(* CODESYS project Full_Project.export

Project tree, tasks and I/O mapping:
  CODESYS_Control_x86_Arca_Control_SM : CODESYS Control x86 Arca Control SM, 3S - Smart Software Solutions GmbH, version 3.5.8.0
    application Application
      libraries: Standard, * (System); Arca Motion Library, 1.0.4.14 (BonMET); Network, 3.5.7.0 (3S - Smart Software Solutions GmbH)
      task Task (cyclic, interval t#5ms, priority 1) calls Main
      AxisControl/
        data type MutiAxisMoveMethod
        function block AuxAxis_PowerOn [ST]
        function block MultiAxisABSMove [ST]
        function block MultiAxisTorqueLimit [ST]
      Hand_Control_blocks/
        data type Error_Message
        data type Gesture_Type
        data type Grab_Command
        data type Grab_State
        data type PhysicalHandType
        function block Grab_Control [ST]
        function block Grab_Demo [ST]
        function block Hand_Gesture [ST]
        function block Hand_Gesture_Demo [ST]
      IO_Management/
        function block Digital_Input [ST]
        function block Digital_Input_Analog [ST]
        function block Digital_Output [ST]
      TCPIP Control/
        data type Robot_Command_via_tcp
        data type Robot_State
        function block TCPServerConnection [ST]
        function block TCP_Command_Extract_And_Analysis [ST]
      Testment_Cartesian_Laser_Platform_Test/
        program Cartesian_Laser_Circle_Testment [ST]
      Testment_Servo_Function_Test/
        program Servo_Testment_Main [ST]
        function block Testment_Message_Manager [ST]
      Utility_functions/
        function block Value_Clamp [ST]
      global variables GLobal_Value
      program Cartesin [ST]
      program Main [ST]
      program Read_Basic_Info [ST]
      program SingleAxis [ST]
    SoftMotion General Axis Pool
*)

// CODESYS_Control_x86_Arca_Control_SM/Application/AxisControl/MutiAxisMoveMethod
TYPE MutiAxisMoveMethod :
(
	None := 0				// all axis move at same vel as given
	, SpeedControl := 10		// all axis arrive destination at same time
);
END_TYPE

// CODESYS_Control_x86_Arca_Control_SM/Application/Hand_Control_blocks/Error_Message
{attribute 'qualified_only'}
{attribute 'strict'}
TYPE Error_Message :
(
	Err_None := 0,
	
	Err_AuxAxis_Movement_Cannot_read_virture_robot_position := 10,	// gesture block not reading robot position
	Err_Gesture_Type_Hand_Pos_Not_Given := 20,	// gesture block not given position
	Err_AuxAxis_Movement_Block_err := 30,	// gesture block first reset movement block err
	Err_Gesture_Type_Cycle_mov_block_err := 40,	// gesture block cycle movement block err
	
	Err_PowerOn_Block_Err := 50,
	Err_PowerOn_TimeOut := 51,
	
	Err_Power_Reset_Block_Err := 60,
	Err_Power_Reset_TimeOut := 61,
	
	Err_Group_Enable_Block_Err := 70,
	Err_Group_Enable_TimeOut := 71
);
END_TYPE

// CODESYS_Control_x86_Arca_Control_SM/Application/Hand_Control_blocks/Gesture_Type
{attribute 'qualified_only'}
{attribute 'strict'}
TYPE Gesture_Type :
(
	Gesture_Type_None			:= 0,
	Gesture_Type_Num_1		:= 1,
	Gesture_Type_Num_2		:= 2,
	Gesture_Type_Num_3		:= 3,
	Gesture_Type_Num_4		:= 4,
	Gesture_Type_Num_5		:= 5,
	Gesture_Type_Num_6		:= 6,
	Gesture_Type_Fist			:= 10,
	Gesture_Type_Palm			:= 11,
	Gesture_Type_ThumbUp		:= 12,
	Gesture_Type_NoNoNo			:= 13,
	Gesture_Type_ComeOnBaby	:= 14,
	Gesture_Type_FingerWave		:= 15,
	Gesture_Type_Wave			:= 16,
	Gesture_Type_Nya			:= 17,
	Gesture_Type_MovObj			:= 18
);
END_TYPE

// CODESYS_Control_x86_Arca_Control_SM/Application/Hand_Control_blocks/Grab_Command
TYPE Grab_Command :
STRUCT
	Tip_Angle : REAL;
	Root_Angle : REAL;
	Clamp_Angle : REAL;
END_STRUCT
END_TYPE

// CODESYS_Control_x86_Arca_Control_SM/Application/Hand_Control_blocks/Grab_State
TYPE Grab_State :
STRUCT
	Tip_State : BOOL;
	Root_State : BOOL;
	Clamp_Angle : REAL;
END_STRUCT
END_TYPE

// CODESYS_Control_x86_Arca_Control_SM/Application/Hand_Control_blocks/PhysicalHandType
TYPE PhysicalHandType :
(
	motor18		:= 0	// total 18 motors. 4 axis for thumb, 3 axis control 2 joints, anohter one control thumb tip joint. Other fingers has 3 axis each, each axis control 1 jonit. 2 axis for each wrist joint.
	, motor17	:= 10	// total 17 motors, each axis control 1 joint.
);
END_TYPE

// CODESYS_Control_x86_Arca_Control_SM/Application/TCPIP Control/Robot_Command_via_tcp
TYPE Robot_Command_via_tcp :
STRUCT
	X_Axis_Valid : BOOL;
	X_value : REAL;
	Y_Axis_Valid : BOOL;
	Y_value : REAL;
	Z_Axis_Valid : BOOL;
	Z_value : REAL;
	Spin : BOOL;
	Grab_Valid : BOOL;
	Grab_state : BOOL := FALSE;
	Gesture_Valid : BOOL;
	Gesture_Num : Gesture_Type;
	Enabl_Hand_Valid : BOOL;
	Enabl_Hand_state : BOOL;
	Gesture_Demo_Valid : BOOL;
	Gesture_Demo_state : BOOL;
	CNC_Mov_Valid : BOOL;
	CNC_Mov_Program_Num : INT;
END_STRUCT
END_TYPE

// CODESYS_Control_x86_Arca_Control_SM/Application/TCPIP Control/Robot_State
TYPE Robot_State :
STRUCT
	Hand_Enabled : BOOL;
	Hand_Enb_Err : BOOL;
	Grab_State : BOOL;
	Gesture_State : Gesture_Type := gesture_type.Gesture_Type_None;
	Hand_Mov_Err : BOOL;
	Robot_Mov_Err : BOOL;
	CNC_Executing : BOOL;
	CNC_Execute_Done : BOOL;
	CNC_Execute_Err : BOOL;
END_STRUCT
END_TYPE

// CODESYS_Control_x86_Arca_Control_SM/Application/GLobal_Value
VAR_GLOBAL
	AllAxisGroupEnb : BOOL;
	Num_of_Axis_GV:WORD;
	Num_of_Groups_GV:WORD;
	Num_of_Cams_GV:WORD;
	MotionCfgOK_GV: BOOL;
	ECatCfgOk_GV: BOOL;
	VisionCfgOk_GV: BOOL;
END_VAR

// CODESYS_Control_x86_Arca_Control_SM/Application/Main
PROGRAM Main
VAR
END_VAR

Read_Basic_Info();

SingleAxis();

Cartesin();

Servo_Testment_Main();

END_PROGRAM

// CODESYS_Control_x86_Arca_Control_SM/Application/Read_Basic_Info
PROGRAM Read_Basic_Info
VAR	
	// read cfg message
	ReadCfg : ArcaLibrary.SYS_GetConfigInfo;
END_VAR

// read how many axis has been config, all *_GV value is golbal value
ReadCfg(axisnumber => Num_of_Axis_GV, groupnumber => Num_of_Groups_GV, cameranumber => Num_of_Cams_GV
	, MotionCfgOk => MotionCfgOK_GV, ecatcfgok => ECatCfgOk_GV, visioncfgok => VisionCfgOk_GV);

END_PROGRAM

// CODESYS_Control_x86_Arca_Control_SM/Application/SingleAxis
PROGRAM SingleAxis
VAR
	Enable : BOOL;
	StartMov : BOOL;
	MovAxis : INT := 0;
	FirstPos : REAL := -180;
	SecondPos : REAL := 180;
	CurrentPos : REAL;
	Vel : REAL := 180;
	Acc : REAL := 180;
	Jerk : REAL := 180;
	stopTime : TIME := T#1S;
	MovErr : BOOL;
	
	PowBlk : ArcaLibrary.MC_Power;
	PowDone, PowErr : BOOL;
	
	MovState : INT;
	FirMov : ArcaLibrary.MC_MoveAbsolute;
	SecMov : ArcaLibrary.MC_MoveAbsolute;
	StopMov : ArcaLibrary.MC_Stop;
	dis_trig : r_trig;
	
	ReadPos : ArcaLibrary.MCAT_ReadAxisMeasures;
	StopTimer : ton;
END_VAR


PowBlk(Axis := MovAxis, Enable:=Enable, EnablePositive:=TRUE, EnableNegative:=TRUE, Status=>PowDone, Error=>PowErr);
ReadPos(axis := MovAxis, enable := PowBlk.Status, pos=> currentPos);

dis_trig(clk := NOT startMov);
StopMov(axis := MovAxis, execute := dis_trig.Q, Deceleration := acc*10, jerk := jerk*10);

IF MovState > 20 AND NOT startMov THEN
	MovState := 20;
END_IF
CASE MovState OF
	0:
		IF PowDone THEN
			MovState := 10;
		END_IF
	10:
		IF startMov THEN
			MovState := 20;
		END_IF
	20:
		FirMov(axis := MovAxis, Execute := FALSE);
		SecMov(axis := MovAxis, Execute := FALSE);
		IF startMov THEN
			StopTimer(in:= FALSE);
			MovState := 30;
		ELSE
			MovState := 0;
		END_IF
	30:
		FirMov(axis := MovAxis, Execute := TRUE, Position := FirstPos
			, Velocity := vel, Acceleration := acc, Deceleration := Acc, jerk := jerk
			, Direction := mcShortestWay, BufferMode := mcAborting 
			, Error => MovErr);
		IF FirMov.Done THEN
			IF stopTime > T#0S THEN
			StopTimer (in := TRUE, PT := stopTime);
				MovState := 35;
			ELSE
				MovState := 40;
			END_IF
		END_IF
	35:
		StopTimer (in := TRUE, PT := stopTime);
		IF StopTimer.Q THEN
			StopTimer(in:= FALSE);
			MovState := 40;
		END_IF
	40:
		SecMov(axis := MovAxis, Execute := TRUE, Position := SecondPos
			, Velocity := vel, Acceleration := acc, Deceleration := Acc, jerk := jerk
			, Direction := mcShortestWay, BufferMode := mcAborting 
			, Error => MovErr);
		IF SecMov.Done THEN
			StopTimer (in := TRUE, PT := stopTime);
			IF stopTime > T#0S THEN
				MovState := 45;
			ELSE
			MovState := 20;
			END_IF
		END_IF
	45:
		StopTimer (in := TRUE, PT := stopTime);
		IF StopTimer.Q THEN
			StopTimer(in:= FALSE);
			MovState := 20;
		END_IF
END_CASE

END_PROGRAM

// CODESYS_Control_x86_Arca_Control_SM/Application/Cartesin
PROGRAM Cartesin
VAR
	Enable : BOOL;
	StartMov : BOOL;
	safe_pos :  ARRAY [1..6] OF REAL := [0.0, 0.0, 0.0, 0.0, -90.0, 0.0];
	FirstReachPos :  ARRAY [1..6] OF REAL := [0.562, 0.333, 0.606, 118.70, 167.069, -70.06];
	SecondReachPos :  ARRAY [1..6] OF REAL := [0.562, 0.3, 0.606, 118.70, 167.069, -70.06];
	FirstPerPos :  ARRAY [1..6] OF REAL := [0.562, 0.333, 0.636, 118.70, 167.069, -70.06];
	SecondPerPos :  ARRAY [1..6] OF REAL := [0.562, 0.3, 0.636, 118.70, 167.069, -70.06];
	
	CurrentPos : REAL;
	Vel : REAL := 10;
	Acc : REAL := 10;
	Jerk : REAL := 10;
	safepoint_overfeed : INT := 5; 
	GrRelCorner :REAL := 0.5;
	MovGroup : INT := 0;
	
	MovErr : BOOL;
	
	PowBlk : AuxAxis_PowerOn;
	PowDone, PowErr : BOOL;
	
	MovState : INT;
	InitialMov : ArcaLibrary.MCAT_MoveDirect;;
	Movs : ARRAY [0..6] OF ArcaLibrary.MC_MoveLinearAbsolute;
	StopMov : ArcaLibrary.MC_GroupStop;
	dis_trig : r_trig;
	
	
END_VAR

PowBlk(Enable := enable, done => PowDone);

dis_trig(clk := NOT startMov);
StopMov(AxesGroup := MovGroup, execute := dis_trig.Q, Deceleration := acc, jerk := jerk, BufferMode := mcAborting);

IF MovState > 20 AND NOT startMov THEN
	MovState := 20;
END_IF
CASE MovState OF
	0:
		IF PowDone THEN
			MovState := 10;
		END_IF
	10:
		IF startMov THEN
			MovState := 20;
		END_IF
	20:
		InitialMov(axesgroup := MovGroup, execute := FALSE);
		Movs[0](axesgroup := MovGroup, Execute := FALSE);
		Movs[1](axesgroup := MovGroup, Execute := FALSE);
		Movs[2](axesgroup := MovGroup, Execute := FALSE);
		Movs[3](axesgroup := MovGroup, Execute := FALSE);
		Movs[4](axesgroup := MovGroup, Execute := FALSE);
		Movs[5](axesgroup := MovGroup, Execute := FALSE);
		IF startMov THEN
			MovState := 30;
		ELSE
			MovState := 0;
		END_IF
	30:
		InitialMov(axesgroup := MovGroup, execute := TRUE, position := ADR(safe_pos), coordsystem := mcacs
			, BufferMode:=mcAborting, TransitionMode:= tmNone, TransitionParameter:= ADR(GrRelCorner) 
			, OverFeedPerc:= safepoint_overfeed);
		IF initialmov.Done THEN
			MovState := 40;
		END_IF
	40:
		IF Movs[4].Done THEN
			Movs[5](axesgroup := MovGroup, Execute := TRUE, Position := ADR(SecondPerPos)
				, Velocity := vel, Acceleration := acc, Deceleration := Acc, jerk := jerk
				, coordsystem := mcMcs, BufferMode := mcBlendingNext
				, TransitionMode := TMcornerdistance, TransitionParameter:=ADR(GrRelCorner)
				, Error => MovErr);
		END_IF
		Movs[0](axesgroup := MovGroup, Execute := TRUE, Position := ADR(FirstPerPos)
			, Velocity := vel, Acceleration := acc, Deceleration := Acc, jerk := jerk
			, coordsystem := mcMcs, BufferMode := mcBlendingNext
			, TransitionMode := TMcornerdistance, TransitionParameter:=ADR(GrRelCorner)
			, Error => MovErr);
		Movs[1](axesgroup := MovGroup, Execute := TRUE, Position := ADR(FirstReachPos)
			, Velocity := vel, Acceleration := acc, Deceleration := Acc, jerk := jerk
			, coordsystem := mcMcs, BufferMode := mcBlendingPrev
			, TransitionMode := TMcornerdistance, TransitionParameter:=ADR(GrRelCorner)
			, Error => MovErr);
		IF Movs[1].Done THEN
			Movs[2](axesgroup := MovGroup, Execute := FALSE);
			Movs[3](axesgroup := MovGroup, Execute := FALSE);
			Movs[4](axesgroup := MovGroup, Execute := FALSE);
			MovState := 50;
		END_IF
	50:
		Movs[2](axesgroup := MovGroup, Execute := TRUE, Position := ADR(FirstPerPos)
			, Velocity := vel, Acceleration := acc, Deceleration := Acc, jerk := jerk
			, coordsystem := mcMcs, BufferMode := mcBlendingNext
			, TransitionMode := TMcornerdistance, TransitionParameter:=ADR(GrRelCorner)
			, Error => MovErr);
		Movs[3](axesgroup := MovGroup, Execute := TRUE, Position := ADR(SecondPerPos)
			, Velocity := vel, Acceleration := acc, Deceleration := Acc, jerk := jerk
			, coordsystem := mcMcs, BufferMode := mcBlendingNext
			, TransitionMode := TMcornerdistance, TransitionParameter:=ADR(GrRelCorner)
			, Error => MovErr);
		Movs[4](axesgroup := MovGroup, Execute := TRUE, Position := ADR(SecondReachPos)
			, Velocity := vel, Acceleration := acc, Deceleration := Acc, jerk := jerk
			, coordsystem := mcMcs, BufferMode := mcBlendingPrev
			, TransitionMode := TMcornerdistance, TransitionParameter:=ADR(GrRelCorner)
			, Error => MovErr);
		IF Movs[4].Done THEN
			Movs[0](axesgroup := MovGroup, Execute := FALSE);
			Movs[1](axesgroup := MovGroup, Execute := FALSE);
			Movs[5](axesgroup := MovGroup, Execute := FALSE);
			MovState := 40;
		END_IF
END_CASE

END_PROGRAM

// CODESYS_Control_x86_Arca_Control_SM/Application/AxisControl/AuxAxis_PowerOn
FUNCTION_BLOCK AuxAxis_PowerOn
VAR_INPUT
	Enable : BOOL;
END_VAR
VAR_OUTPUT
	Done : BOOL;
	Error : BOOL;
	Err_Message : Error_Message;
END_VAR
VAR
	_state : INT := 0;
	_end : BOOL := TRUE;
	_Timer: ton;
	_err_time : TIME := T#5S;
	
	// read cfg message
	ReadCfg : ArcaLibrary.SYS_GetConfigInfo;
	Num_of_Axis:WORD;
	Num_of_Groups:WORD;
	Num_of_Cams:WORD;
	MotionCfgOK: BOOL;
	ECatCfgOk: BOOL;
	VisionCfgOk: BOOL;
	
	// power settings
	PowBlk:ARRAY[1..48] OF ArcaLibrary.MC_Power;
	PowDone, PowErr: ARRAY [1..48] OF BOOL;
	power_On_States : INT := 0;
	All_Power_On_Check_Counter : INT;
	Power_Err_Check_Counter : INT;
	Power_Counter : INT;
	
	//reset blocks
	AxRes:ARRAY[1..48] OF ArcaLibrary.MC_Reset;
	AxResDone, AxResErr: ARRAY [1..48] OF BOOL;
	rest_counter : INT := 0;
	All_reset_On : BOOL;
	All_reset_On_Check_Counter : INT;
	reset_Err_Check_Counter : INT;
	reset_State : INT := 0;
	
	//group management
	GrpEn: ARRAY[1..5] OF ArcaLibrary.MC_GroupEnable;
	GrpDis: ARRAY[1..5] OF ArcaLibrary.MC_GroupDisable;
	GrpErr : ARRAY [1..5] OF BOOL;
	Grp_En_State : INT;
	Grp_counter : INT;
	Grp_En_Check_Counter : INT;
	Grp_Dis_Counter : INT;
	
	//debug
END_VAR

IF enable  THEN
	_end := FALSE;
ELSE
	_state := -10;
END_IF

IF _end = TRUE THEN
	RETURN;
END_IF

_Timer(in:= (power_On_States = 10) OR (reset_State = 10) OR (Grp_En_State = 10), pt:= _err_time);

// read how many axis has been config
ReadCfg(axisnumber => Num_of_axis, groupnumber => Num_of_Groups, cameranumber => Num_of_Cams
	, MotionCfgOk => MotionCfgOK, ecatcfgok => ECatCfgOk, visioncfgok => VisionCfgOk);

// power blocks
CASE (power_On_States) OF
	0:	
		IF (_state>0 AND _state<100) AND ECatCfgOk AND MotionCfgOK THEN
			power_On_States := 10;
		END_IF
	10:
		All_Power_On_Check_Counter := 1;
		FOR Power_Counter:=1 TO WORD_TO_INT(Num_of_axis) DO
			PowBlk[Power_Counter](Axis:=Power_Counter -1, Enable:=TRUE, EnablePositive:=TRUE, EnableNegative:=TRUE, Status=>PowDone[Power_Counter], Error=>PowErr[Power_Counter]);
			IF PowDone[Power_Counter] = TRUE THEN
				All_Power_On_Check_Counter := All_Power_On_Check_Counter + 1;
			END_IF
		END_FOR
		
		IF All_Power_On_Check_Counter >= WORD_TO_INT(Num_of_axis) THEN
			power_On_States := 20;
		ELSIF _Timer.Q THEN
			_state := -21;
		END_IF
		IF (_state<=0 OR _state>=100) THEN
			power_On_States := 30;
		END_IF
	20:
		IF (_state<=0 OR _state>=100) THEN
			power_On_States := 30;
		END_IF
	30:
		FOR Power_Counter:=1 TO WORD_TO_INT(Num_of_axis) DO
			PowBlk[Power_Counter](Axis:=Power_Counter -1, Enable:=FALSE);
		END_FOR
		power_On_States := 0;
END_CASE
// check if power block is err
IF power_On_States > 0 AND power_On_States < 30 THEN
	FOR Power_Err_Check_Counter:=1 TO WORD_TO_INT(Num_of_axis) DO
			IF PowBlk[Power_Err_Check_Counter - 1].Error = TRUE THEN
				//_state := -20;
			END_IF
	END_FOR
END_IF

// reset blocks
CASE (reset_State) OF
	0:
		All_reset_On := FALSE;
		IF _state=2 THEN
			reset_state := 10;
		END_IF
	10:
		All_reset_On_Check_Counter := 0;
		FOR rest_counter:=1 TO WORD_TO_INT(Num_of_axis) DO
			AxRes[rest_counter](Axis:=rest_counter - 1, Execute:=TRUE, Done=>AxResDone[rest_counter], Error=>AxResErr[rest_counter]);
			IF AxRes[rest_counter].Done = TRUE THEN
				All_reset_On_Check_Counter := All_reset_On_Check_Counter +1;
			END_IF
		END_FOR
		IF All_reset_On_Check_Counter = WORD_TO_INT(Num_of_axis) THEN
			All_reset_On := TRUE;
		ELSIF _Timer.Q THEN
			_state := -31;
		END_IF
		IF (_state <> 2) THEN
			reset_State := 0;
		END_IF
END_CASE
// check if reset block is err
IF reset_State <> 0 THEN
	FOR reset_Err_Check_Counter:=1 TO WORD_TO_INT(Num_of_axis) DO
			IF AxRes[reset_Err_Check_Counter - 1].Error = TRUE THEN
				_state := -30;
			END_IF
	END_FOR
END_IF

// group enable/disable
CASE Grp_En_State OF
	0:
		IF _state >= 30 AND _state <=100 THEN
			grp_counter := 1;
			Grp_En_State := 10;
		END_IF
	10:	
		IF grp_counter > WORD_TO_INT(Num_of_Groups) THEN
			Grp_En_State := 20;
		ELSE
			GrpEn[grp_counter](AxesGroup := grp_counter - 1, Execute := TRUE);
			IF GrpEn[grp_counter].Done THEN
				IF grp_counter <= WORD_TO_INT(Num_of_Groups) THEN
					grp_counter := grp_counter +1;
				END_IF
			ELSIF _Timer.Q THEN
				_state := -41;
			END_IF
		END_IF
		
		IF (_state < 30 OR _state > 100) THEN
			Grp_En_State := 30;
		END_IF
	20:
		IF (_state < 30 OR _state > 100) THEN
			Grp_En_State := 30;
		END_IF
	30:
		FOR grp_counter := 1 TO WORD_TO_INT(Num_of_Groups) DO
			GrpEn[grp_counter](AxesGroup := grp_counter - 1, Execute := FALSE);
		END_FOR
		Grp_En_State := 0;
	
END_CASE
// check if enable block is err
IF Grp_En_State = 9990 THEN
	FOR Grp_En_Check_Counter:=1 TO WORD_TO_INT(Num_of_Groups) DO
			IF GrpEn[Grp_En_Check_Counter - 1].Error = TRUE THEN
				_state := -40;
			END_IF
	END_FOR
END_IF

// disable group when all group enable block are off
FOR Grp_Dis_Counter := 1 TO WORD_TO_INT(Num_of_Groups) DO
	GrpDis[Grp_Dis_Counter](AxesGroup:= Grp_Dis_Counter - 1, Execute:= Grp_En_State = 0);
END_FOR

//	manager
CASE _state OF
	-41:
		error := TRUE;
		err_message := Error_Message.Err_Group_Enable_TimeOut;
	-40:
		error := TRUE;
		err_message := Error_Message.Err_Group_Enable_Block_Err;
		
	-31:
		error := TRUE;
		err_message := Error_Message.Err_Power_Reset_TimeOut;
	-30:
		error := TRUE;
		err_message := Error_Message.Err_Power_Reset_Block_Err;
		
	-21:
		error := TRUE;
		err_message := Error_Message.Err_PowerOn_TimeOut;
	-20:
		error := TRUE;
		err_message := Error_Message.Err_PowerOn_Block_Err;
	-10:
		IF power_On_States = 0 AND reset_State = 0 AND Grp_En_State = 0 THEN
			done := error := FALSE;
			err_message := error_message.Err_None;
			_end := TRUE;
			_state := 0;
		END_IF
	0:
		IF enable AND power_On_States = 0 AND reset_State = 0 AND Grp_En_State = 0 THEN
			_state := 10;
		END_IF
	10:
		IF power_On_States = 20 THEN
			_state := 30;
		END_IF
	30:
		IF Grp_En_State = 20 THEN
			_state := 40;
		END_IF
	40:
		done := TRUE;
END_CASE

END_FUNCTION_BLOCK

// CODESYS_Control_x86_Arca_Control_SM/Application/Testment_Servo_Function_Test/Servo_Testment_Main
PROGRAM Servo_Testment_Main
VAR
	Set_Do: ARRAY [1..8] OF BOOL;
	Read_DI: ARRAY [1..12] OF BOOL;
	Read_DIA_Percentage :  ARRAY [0..7] OF REAL;
	Read_DIA_Raw :  ARRAY [0..7] OF UINT;
	
	// axis define
	FirstAxis : WORD := 1;
	LastAxis : WORD := 6;	// this value has been automaticlly asigned by global config reader
	//DI
	DI_Block : Digital_Input;
	
	//DO
	DO_Block : Digital_Output;
	
	//DIA
	smTime : TIME := T#250MS;
	DIA_Block : Digital_Input_Analog;
	
	
	// Testment functions
	Servo_Testment_State : INT := -1;
	Test_Process_Start_Restart, Error_State : BOOL;
	Message_Manager : Testment_Message_Manager;
	Show_Text : WSTRING;
	enb_axis : AuxAxis_PowerOn;
	read_axis : ARRAY [1..6] OF Arcalibrary.MCAT_ReadAxisMeasures;
	home_axis : ARRAY [1..6] OF Arcalibrary.MC_Home;
	re_j : INT;
	ts_i: INT;
	timer : ton;
	check_pos_err : REAL := 5;
	
	mov_axis : ARRAY [1..6] OF ArcaLibrary.MC_MoveAbsolute;
	FirstPos : REAL := 360;
	SecondPos : REAL := -360;
	CurrentPos : REAL;
	Vel : REAL := 180;
	Acc : REAL := 1900;
	Jerk : REAL := 9500;
	axis_mov_counter : INT;
	
	analog_cap ,analog_base : ARRAY [0..7] OF UINT;
	analog_difference : UINT := 12500; // 5v should be around 12900 ~ 13000
	set_override : ArcaLibrary.MC_GroupSetOverride;
	set_limit : ArcaLibrary.MCAT_AxisSetLimits;
	// analog control motor speed function
	analog_motor_state :INT := -1;
	debugButton : BOOL;
	speedLimit : REAL;
	analogFirPos : REAL := 380;
	analogSecPos : REAL := -380;
	analogVel : REAL := 18000;
	analogACC : REAL := 900000;
	analogJerk : REAL := 45000000;
	(* legacy ------
	forCounter: INT;
	//DI
	Read_6Ax_DI: Arcalibrary.ECAT_GetPdi_U32;
	DI_Raw : UDINT;
	new_DI_Value : UINT;
	
	//DO
	new_Do_Value, old_Do_Value : UINT;
	Write_6Ax_Do: Arcalibrary.ECAT_SetPdo_U32;
	------*)
	
	// servo elder program
	servo_elder_state :INT := -1;
	// elder_MoveType
	// 0 msans postion control all axis stop and turn in same time
	// 1 means speed control, two groups stop and turn in different times
	elder_MoveType : WORD := 1;
	elderVel : REAL := 18000;
	elderACC : REAL := 900000;
	elderJerk : REAL := 45000000;
	el_i : INT;
	speedFirGroup : ARRAY [0..5] OF ArcaLibrary.MC_MoveVelocity;
	speedSecGroup : ARRAY [0..5] OF ArcaLibrary.MC_MoveVelocity;
	elderTimer : ton;
	speedGroupSwitch : BOOL;
	speedSwitchTime : TIME := T#50MS;
	speedFirDir : ArcaLibrary.mc_Direction := mcPositiveDirection;
	speedSecDir : ArcaLibrary.mc_Direction := mcNegativeDirection;
	
	// 6 axis io test
	try: UINT;
	try2 : REAL;
	try3 : REAL := 3.9;
	read_0 : UINT;
	read_1 : UDINT;
	read_2 :ULINT;
	andValue : WORD;
	switch : BOOL;
	offsetValue : WORD := 147;
	TestAin_0: Arcalibrary.ECAT_GetPdi_U16;
	TestAin_1: Arcalibrary.ECAT_GetPdi_U32;
	TestAin_2: Arcalibrary.ECAT_GetPdi_U64;
	MaxmentOffset : UINT := 50;
	found_0, found_1, found_2, starter, maunl_next : BOOL;
	target_low : UINT := 12700;
	target_high : UINT := 13000;
	
	debugTimer : ton;
	FirstReachPos :  ARRAY [1..6] OF REAL := [0.6, -0.2, 0.606, -31.346, 178.434, 149.160];
	SecondReachPos :  ARRAY [1..6] OF REAL := [0.6, 0.2, 0.606, -31.346, 178.434, 149.160];
	Vell : REAL := 10;
	Accl : REAL := 10;
	Jerkl : REAL := 10;
	GrRelCorner :REAL := 0.5;
	MovErr : BOOL;
	//Movs : ARRAY [0..6] OF ArcaLibrary.MC_MoveLinearAbsolute;
	
	// error light control
	ErrLightControlState : INT;
	ErrLightTimer : Ton;
	ErrLightBlinkTime : TIME := T#200MS;
	ErrLightFinishTime : TIME := T#500MS;
	ErrLightCounterHigh : INT;
	ErrLightCounterLow : INT;
	ErrLight_i : INT;
	ErrLight_Switch : BOOL;
	// debug
	// --- because of homing bug (new servo need to home twice), get some function foe step 30
	homeErrOnce : BOOL;
	//---
	
	// debug
	manual_m01 : BOOL;
	manual_00 : BOOL;
	manual_20 : BOOL;
	manual_50 : BOOL;
	manual_jump_analog_check : BOOL;
	
	// debug para start---------------------------
	// read cfg message
	ReadCfg : ArcaLibrary.SYS_GetConfigInfo;
	Num_of_Axis:WORD;
	PowerState : ARRAY [0..5] OF ArcaLibrary.MCAT_ReadPowerStatus;
	AxisMeasure : ARRAY [0..5] OF ArcaLibrary.MCAT_ReadAxisMeasures;
	cfg_i : INT;
	
	//speed control test
	SC_Enb : BOOL; 
	SCMovTime : TIME := T#500MS;
	SCTimer : TON;
	SC_State : INT;
	SC_i,SC_y : INT;
	SpeedMovFir : ARRAY [0..5] OF ArcaLibrary.MC_MoveVelocity;
	SpeedMovSec : ARRAY [0..5] OF ArcaLibrary.MC_MoveVelocity;
	SCVel : REAL := 1800;
	SCACC : REAL := 9000;
	SCJerk : REAL := 45000;
	SCFirDir : ArcaLibrary.mc_Direction := mcPositiveDirection;
	SCSecDir : ArcaLibrary.mc_Direction := mcNegativeDirection;
	SCGroupSwitch : BOOL;
	
	// debug para end-----------------------------------
END_VAR

/////////////////////////////// instruction windows in chinsese  /////////////////////////////////////////

Message_Manager(state_in := Servo_Testment_State
	, start_restart_indicator => Test_Process_Start_Restart
	, Show_Message => Show_Text
	);
	
/////////////////////////////// instruction windows in chinsese  /////////////////////////////////////////

// if ethercat not ready then return
IF NOT ECatCfgok_GV THEN
	DI_Block (enable := FALSE);
	DO_Block (enable := FALSE);
	RETURN;
END_IF

IF Num_of_Axis_GV > 6 THEN
	Servo_Testment_State := -5;
END_IF
LastAxis := Num_of_Axis_GV;

DI_Block(enable := TRUE, DI_Array => Read_DI);
DO_Block(enable := TRUE, DO_Array := Set_Do);
DIA_Block(enable := TRUE, smoothTime := smTime
	, MaxRawInputValue := analog_cap
	, MinRawInputValue := analog_base
	, DIA_Raw => Read_DIA_Raw
	, DIA_Process => Read_DIA_Percentage
	);

enb_axis (enable := Servo_Testment_State > 9);
FOR re_j := 1 TO WORD_TO_INT(Num_of_Axis_GV) DO
	read_axis[re_j](axis := re_j - 1, enable :=  TRUE);
END_FOR

timer(in:= Servo_Testment_State = 30, pt := T#2S);

IF Servo_Testment_State <> -1 AND ((Read_DI[1] AND Read_DI[2]) OR manual_m01) THEN
	Servo_Testment_State := 0;
END_IF


set_limit(execute := debugButton, axis := 0, speedLimit := speedLimit); // useless

IF Servo_Testment_State < 130 THEN
	set_override(axesgroup := 0, enable := TRUE
	, velFactor := 1, accfactor := 1, jerkFactor := 1);
ELSE
	set_override(axesgroup := 0, enable := TRUE
	, velFactor := Read_DIA_Percentage[0]/100
	, accfactor := 1
	, jerkFactor := 1
	);
END_IF

IF Servo_Testment_State = 0 THEN	// reset
	//Set_Do[7]:= TRUE;
	//Set_Do[8]:= TRUE;
	homeErrOnce:= FALSE;
END_IF

CASE Servo_Testment_State OF
	-50: // analog cap and base difference too small
		// please connection and input voltage
		analog_cap[0];	// cap value
		analog_base[0];	// base vaule
	
	-45: // axis not mov to corrent pos
		ts_i; // error axis;
	-40: // if axis get err when moving
		ts_i; // error axis
	
	-35: // if some axis is not near 0 after homing
		ts_i; // error axis
		
	-33: // if some axis home err or time out
		ts_i;	// error axis
		
	-30: // if some axis home err
		home_axis[ts_i].ErrorID;	// homing err message
		
	-20: // if some axis can not enable
		enb_axis.Err_Message;	// enable err message
		
	-10: // if button is not commanding right inputs
		// plz check input button
		
	-5:	// config file contain more than 6 axis and exceed this program can handle
	
	-1:
		IF Read_DI[1] AND Read_DI[2] OR manual_m01 THEN
			Servo_Testment_State:= 0;
		ELSIF  Read_DI[1] OR Read_DI[2] THEN
			Servo_Testment_State := -10;	// if there is any input not receiving signal
		END_IF
		
	0:	// push second button to enable all axis
		IF Read_DI[3] AND Read_DI[4] AND Read_DI[5] AND Read_DI[6] OR manual_00 THEN
			Servo_Testment_State:= 10;
		ELSIF  Read_DI[3] OR Read_DI[4] OR Read_DI[5] OR Read_DI[6] THEN
			Servo_Testment_State := -10;	// if there is any input not receiving signal
		END_IF
	5:	// restart
		Servo_Testment_State := 10;
	10: // if 1~6 input is ok, waitting axis to enable
		IF enb_axis.Done THEN
			Servo_Testment_State := 20; // if enabled
		ELSIF enb_axis.Error THEN
			Servo_Testment_State := -20; // if some axis fail to enable
		END_IF
	20: // push third button to home axis
		FOR ts_i := WORD_TO_INT(FirstAxis) TO WORD_TO_INT(LastAxis) DO
			home_axis[ts_i](axis := ts_i - 1, execute := FALSE);	// reset blocks
		END_FOR
		IF Read_DI[7] AND Read_DI[8] AND Read_DI[9] OR homeErrOnce OR manual_20 THEN
			ts_i:= WORD_TO_INT(FirstAxis);
			Servo_Testment_State := 30;
		ELSIF Read_DI[7] OR Read_DI[8] OR Read_DI[9] THEN
			Servo_Testment_State := -10;	// if there is any input not receiving signal
		END_IF
	30: // start homing axis	// should not use I lkie in this case, is confilc with other state machine
		//Set_Do[7]:= TRUE;
		home_axis[ts_i](axis := ts_i - 1, execute := TRUE, position := 0, buffermode := mcAborting);
		IF home_axis[LastAxis].Done THEN	// all axis according to config file had homed
			FOR ts_i := WORD_TO_INT(FirstAxis) TO WORD_TO_INT(LastAxis) DO
				home_axis[ts_i](axis := ts_i - 1, execute := FALSE);
			END_FOR
			Servo_Testment_State := 40;
		ELSIF home_axis[ts_i].Done AND ts_i <= WORD_TO_INT(LastAxis) THEN // if current axis homing done
			timer(in:= FALSE);	// reset timer
			ts_i := ts_i + 1;
		ELSIF home_axis[ts_i].Error THEN	// if current axis get err
			Servo_Testment_State := -30;
		ELSIF timer.Q THEN	// if current axis not finish homing in certen time
			Servo_Testment_State := -33;
		END_IF
	40: // check if all axis are home
		ts_i := WORD_TO_INT(FirstAxis - 1);
		WHILE (ts_i < WORD_TO_INT(LastAxis)) AND Servo_Testment_State = 40 DO
			ts_i := ts_i + 1;
			IF read_axis[ts_i].Pos > check_pos_err OR read_axis[ts_i].Pos < -check_pos_err THEN // if current axis pos more than check_pos_err
				Servo_Testment_State := -35;
			END_IF
		END_WHILE
		IF Servo_Testment_State <> -35 THEN
			//Set_Do[8]:= TRUE;
			Servo_Testment_State := 50;
		END_IF
	50: // push fourth button to order motor turn
		FOR ts_i := WORD_TO_INT(FirstAxis) TO WORD_TO_INT(LastAxis) DO
			mov_axis[ts_i](axis := ts_i - 1, execute := FALSE);	// reset blocks
		END_FOR
		IF (Read_DI[10] AND Read_DI[11] AND Read_DI[12]) OR homeErrOnce OR manual_50 THEN
			Servo_Testment_State := 60;
		ELSIF Read_DI[10] OR Read_DI[11] OR Read_DI[12] THEN
			Servo_Testment_State := -10;	// if there is any input not receiving signal
		END_IF
	60:
		axis_mov_counter := 0;
		ts_i := WORD_TO_INT(FirstAxis - 1);
		WHILE ts_i < WORD_TO_INT(LastAxis) AND Servo_Testment_State = 60 DO
			ts_i := ts_i + 1;
			mov_axis[ts_i](axis := ts_i - 1, Execute := TRUE, Position := FirstPos
			, Velocity := vel, Acceleration := acc, Deceleration := Acc, jerk := jerk
			, Direction := mcShortestWay, BufferMode := mcAborting
			);
			IF mov_axis[ts_i].Done THEN
				axis_mov_counter := axis_mov_counter + 1;
			ELSIF  mov_axis[ts_i].Error THEN
				Servo_Testment_State := -40;	// axis err when moving
				IF NOT homeErrOnce THEN
					homeErrOnce := TRUE;
					Servo_Testment_State := 5;	// give secend chance
				END_IF
			END_IF
		END_WHILE
		IF axis_mov_counter >= WORD_TO_INT(LastAxis - (FirstAxis - 1)) AND Servo_Testment_State <> -40 THEN // if all axis mov done
			FOR ts_i := WORD_TO_INT(FirstAxis) TO WORD_TO_INT(LastAxis) DO
				mov_axis[ts_i](axis := ts_i - 1, execute := FALSE);	// reset blocks
			END_FOR
			Servo_Testment_State := 70;
		END_IF
	70: // check pos
		ts_i :=  WORD_TO_INT(FirstAxis - 1);
		WHILE ts_i < WORD_TO_INT(LastAxis) AND Servo_Testment_State = 70 DO
			ts_i := ts_i + 1;
			IF FirstPos - read_axis[ts_i].Pos < -check_pos_err OR FirstPos - read_axis[ts_i].Pos > check_pos_err THEN // if current axis pos more than check_pos_err
				Servo_Testment_State := -45;
			END_IF
		END_WHILE
		
		IF Servo_Testment_State <> -45 THEN
			Servo_Testment_State := 80;
		END_IF
		
	80: // motor start to turn
		axis_mov_counter := 0;
		ts_i := FirstAxis - 1;
		WHILE ts_i < WORD_TO_INT(LastAxis) AND Servo_Testment_State = 80 DO
			ts_i := ts_i + 1;
			mov_axis[ts_i](axis := ts_i - 1, Execute := TRUE, Position := SecondPos
			, Velocity := vel, Acceleration := acc, Deceleration := Acc, jerk := jerk
			, Direction := mcShortestWay, BufferMode := mcAborting
			);
			IF mov_axis[ts_i].Done THEN
				axis_mov_counter := axis_mov_counter + 1;
			ELSIF  mov_axis[ts_i].Error THEN
				Servo_Testment_State := -40;	// axis err when moving
			END_IF
		END_WHILE
		IF axis_mov_counter >= LastAxis - (FirstAxis - 1) AND Servo_Testment_State <> -40 THEN // if all axis mov done
			Servo_Testment_State := 90;
		END_IF
		
	90: // check pos
		ts_i := FirstAxis - 1;
		WHILE ts_i < WORD_TO_INT(LastAxis) AND Servo_Testment_State = 90 DO
			ts_i := ts_i + 1;
			IF SecondPos - read_axis[ts_i].Pos < -check_pos_err OR SecondPos - read_axis[ts_i].Pos > check_pos_err THEN // if current axis pos more than check_pos_err
				Servo_Testment_State := -45;
			END_IF
		END_WHILE
		IF Servo_Testment_State <> -45 THEN
			FOR ts_i := WORD_TO_INT(FirstAxis) TO WORD_TO_INT(LastAxis) DO
				mov_axis[ts_i](axis := ts_i - 1, execute := FALSE);	// reset blocks
			END_FOR
			Servo_Testment_State := 100;
		END_IF
		
	100: // set analog input base value, click second button to remember
		analog_base[0] := Read_DIA_Raw[0];
		IF Read_DI[3] AND Read_DI[4] AND Read_DI[5] AND Read_DI[6] OR manual_jump_analog_check THEN
			Servo_Testment_State:= 110;
		ELSIF  Read_DI[3] OR Read_DI[4] OR Read_DI[5] OR Read_DI[6] THEN
			Servo_Testment_State := -10;	// if there is any input not receiving signal
		END_IF
		
	110: // set analog input cap value, click third button to remember
		analog_cap[0] := Read_DIA_Raw[0];
		IF Read_DI[7] AND Read_DI[8] AND Read_DI[9] OR manual_jump_analog_check THEN
			Servo_Testment_State := 120;
		ELSIF Read_DI[7] OR Read_DI[8] OR Read_DI[9] THEN
			Servo_Testment_State := -10;	// if there is any input not receiving signal
		END_IF
		
	120: // check difference between cap and base
		IF (analog_cap[0] - analog_base[0] > analog_difference) OR manual_jump_analog_check THEN
			Servo_Testment_State := 130;
		ELSE
			Servo_Testment_State := -50;
		END_IF
	130:
		
	//100: // procedure done
		
END_CASE

(*IF Servo_Testment_State < 130 THEN
	analog_motor_state := -1;
END_IF

(*************
original Servo_Testment_State > 130 is designed for analog control axis speed
currently this state is use for servo elder testment
*******************)
CASE analog_motor_state	OF

	-1:
		//analog_motor_state := 0;
	0:
		FOR i := 1 TO WORD_TO_INT(Num_of_Axis_GV) DO	// should not use I here because this I is conflic with test state
			mov_axis[i](axis := i - 1, execute := FALSE);	// reset blocks
		END_FOR
		analog_motor_state := 10;
		debugTimer(in:= FALSE);
		(*
	10:
		mov_axis[1](axis := 0, Execute := TRUE, Position := 0);
		mov_axis[2](axis := 1, Execute := TRUE, Position := 0);
		mov_axis[3](axis := 2, Execute := TRUE, Position := 0);
		mov_axis[4](axis := 3, Execute := TRUE, Position := 0);
		mov_axis[5](axis := 4, Execute := TRUE, Position := 0);
		mov_axis[6](axis := 5, Execute := TRUE, Position := 0);
		debugTimer (in:= TRUE, pt := T#5S);
		IF debugTimer.Q THEN
			debugTimer(in:= FALSE);
			
			FOR i := 1 TO WORD_TO_INT(Num_of_Axis_GV) DO
				mov_axis[i](axis := i - 1, execute := FALSE);	// reset blocks
			END_FOR
			analog_motor_state := 20;
			
			Movs[0](axesgroup := 0, Execute := FALSE);
			
			Movs[1](axesgroup := 0, Execute := FALSE);
		END_IF
		
	20:
		Movs[0](axesgroup := 0, Execute := TRUE, Position := ADR(FirstReachPos)
			, Velocity := vell, Acceleration := accl, Deceleration := Accl, jerk := jerkl
			, coordsystem := mcMcs, BufferMode := mcAborting
			, TransitionMode := tmNone, TransitionParameter:=ADR(GrRelCorner)
			, Error => MovErr);
		IF Movs[0].Done THEN
			Movs[0](axesgroup := 0, Execute := FALSE);
			analog_motor_state := 30;
		END_IF
	30:
		Movs[1](axesgroup := 0, Execute := TRUE, Position := ADR(SecondReachPos)
			, Velocity := vell, Acceleration := accl, Deceleration := Accl, jerk := jerkl
			, coordsystem := mcMcs, BufferMode := mcAborting
			, TransitionMode := tmNone, TransitionParameter:=ADR(GrRelCorner)
			, Error => MovErr);
		IF Movs[1].Done THEN
			Movs[1](axesgroup := 0, Execute := FALSE);
			analog_motor_state := 20;
		END_IF
	*)
END_CASE*)

IF Servo_Testment_State < 130 THEN
	servo_elder_state := -1;
END_IF
CASE servo_elder_state OF
	-1:
		IF elder_MoveType = 0 THEN	// if control in abs 
			servo_elder_state := 0;
		ELSIF elder_MoveType = 1 THEN	// if control in vel
			servo_elder_state := 30;
		END_IF
	0:
		FOR el_i := 1 TO WORD_TO_INT(Num_of_Axis_GV) DO
			mov_axis[el_i](axis := el_i - 1, execute := FALSE);	// reset blocks
		END_FOR
		
		servo_elder_state := 10;
	10:
		axis_mov_counter := 0;
		el_i := 0;
		WHILE el_i < WORD_TO_INT(LastAxis - (FirstAxis - 1)) AND Servo_Testment_State <> -40 DO
			el_i := el_i + 1;
			mov_axis[el_i](axis := el_i - 1, Execute := TRUE, Position := analogFirPos
				, velocity := elderVel, Acceleration := elderACC, Deceleration := elderACC, Jerk := elderJerk
				, Direction := mcShortestWay, BufferMode := mcAborting
			);
			IF mov_axis[el_i].Done THEN
				axis_mov_counter := axis_mov_counter + 1;
			ELSIF  mov_axis[el_i].Error THEN
				Servo_Testment_State := -40;	// axis err when moving
			END_IF
		END_WHILE
		IF axis_mov_counter >= 6 AND Servo_Testment_State <> -40 THEN // if all axis mov done
			FOR el_i := WORD_TO_INT(FirstAxis) TO WORD_TO_INT(LastAxis) DO
				mov_axis[el_i](axis := el_i - 1, execute := FALSE);	// reset blocks
			END_FOR
			servo_elder_state := 20;
		END_IF
	20:
		axis_mov_counter := 0;
		el_i := 0;
		WHILE el_i < WORD_TO_INT(LastAxis - (FirstAxis - 1)) AND Servo_Testment_State <> -40 DO
			el_i := el_i + 1;
			mov_axis[el_i](axis := el_i - 1, Execute := TRUE, Position := analogSecPos
				, velocity := elderVel, Acceleration := elderACC, Deceleration := elderACC, Jerk := elderJerk
				, Direction := mcShortestWay, BufferMode := mcAborting
			);
			IF mov_axis[el_i].Done THEN
				axis_mov_counter := axis_mov_counter + 1;
			ELSIF  mov_axis[el_i].Error THEN
				Servo_Testment_State := -40;	// axis err when moving
			END_IF
		END_WHILE
		IF axis_mov_counter >= 6 AND Servo_Testment_State <> -40 THEN // if all axis mov done
			FOR el_i := WORD_TO_INT(FirstAxis) TO WORD_TO_INT(LastAxis) DO
				mov_axis[el_i](axis := el_i - 1, execute := FALSE);	// reset blocks
			END_FOR
			servo_elder_state := 10;
		END_IF
	30:
		FOR el_i := 0 TO 5 DO
			speedFirGroup[el_i](axis := el_i,execute := FALSE);
			speedSecGroup[el_i](axis := el_i,execute := FALSE);
		END_FOR
		elderTimer(in := FALSE);
		speedGroupSwitch := FALSE;
		servo_elder_state := 40;
	40:
		elderTimer(in := TRUE, pt := speedSwitchTime);
		IF elderTimer.Q THEN	// if time reached
			IF NOT speedGroupSwitch THEN	//decide which motor group is time to switch dir
				speedGroupSwitch := TRUE;
				IF speedFirDir = mcPositiveDirection THEN	// if first group is moving positivily
					speedFirDir := mcNegativeDirection;	// then switch to negative
				ELSE
					speedFirDir := mcPositiveDirection;
				END_IF
			ELSE
				speedGroupSwitch := FALSE;
				IF speedSecDir = mcPositiveDirection THEN
					speedSecDir := mcNegativeDirection;
				ELSE
					speedSecDir := mcPositiveDirection;
				END_IF
			END_IF
		END_IF
		FOR el_i := 0 TO 5 BY 2 DO
			speedFirGroup[el_i](axis := el_i,execute := NOT (elderTimer.Q AND speedGroupSwitch)	// only switch off when timer is alarted and first group direction is switched
				, velocity := elderVel, Acceleration := elderACC, Deceleration := elderACC, Jerk := elderJerk
				, Direction := speedFirDir, Buffermode := mcAborting);
			IF  speedFirGroup[el_i].Error THEN
				Servo_Testment_State := -40;	// axis err when moving
			END_IF
		END_FOR
		FOR el_i := 1 TO 5 BY 2 DO
			speedFirGroup[el_i](axis := el_i,execute := NOT (elderTimer.Q AND NOT speedGroupSwitch)	// only switch off when timer is alarted and second group direction is switched
				, velocity := elderVel, Acceleration := elderACC, Deceleration := elderACC, Jerk := elderJerk
				, Direction := speedSecDir, Buffermode := mcAborting);
			IF  speedFirGroup[el_i].Error THEN
				Servo_Testment_State := -40;	// axis err when moving
			END_IF
		END_FOR
		
		IF elderTimer.Q THEN	// if time reached
			elderTimer(in := FALSE);	// switch off timer
		END_IF
END_CASE

IF Servo_Testment_State > -1 THEN
	errlightcontrolstate := 0;
END_IF
CASE errlightcontrolstate OF
	0:
		Set_Do[7]:= TRUE;
		Set_Do[8]:= TRUE;
		IF Servo_Testment_State < 0 THEN
			Set_Do[7]:= FALSE;
			Set_Do[8]:= FALSE;
			ErrLightCounterHigh := (ABS(Servo_Testment_State) / 10) MOD 10;
			ErrLightCounterLow := ABS(Servo_Testment_State) MOD 10;
			ErrLightTimer(in := FALSE);
			ErrLight_i := 0;
			ErrLight_Switch := FALSE;
			IF ErrLightCounterHigh > 0 THEN
				errlightcontrolstate := 10;	// if there have higer num next state
			ELSE
				errlightcontrolstate := 20;	// go to low num directily
			END_IF
		END_IF
	10:	// blink higher number
		Set_Do[7]:= ErrLight_Switch;
		ErrLightTimer(in := TRUE , pt:= ErrLightBlinkTime);
		IF ErrLightTimer.Q THEN
			IF ErrLight_Switch THEN
				ErrLight_Switch := FALSE;
			ELSE
				ErrLight_Switch := TRUE;
			END_IF
			ErrLightTimer (in := FALSE);
			ErrLight_i := ErrLight_i + 1;
		END_IF
		IF ErrLight_i >= (ErrLightCounterHigh * 2) THEN
			ErrLightTimer(in := FALSE);
			ErrLight_i := 0;
			ErrLight_Switch := FALSE;
			IF ErrLightCounterLow > 0 THEN
				errlightcontrolstate := 20;	// if have lower num
			ELSE
				errlightcontrolstate := 30;	// go wating time
			END_IF
		END_IF
	20:// blink lower number
		Set_Do[8]:= ErrLight_Switch;
		ErrLightTimer(in := TRUE , pt:= ErrLightBlinkTime);
		IF ErrLightTimer.Q THEN
			IF ErrLight_Switch THEN
				ErrLight_Switch := FALSE;
			ELSE
				ErrLight_Switch := TRUE;
			END_IF
			ErrLightTimer (in := FALSE);
			ErrLight_i := ErrLight_i + 1;
		END_IF
		IF ErrLight_i >= (ErrLightCounterLow * 2) THEN
			ErrLightTimer(in := FALSE);
			ErrLight_i := 0;
			ErrLight_Switch := FALSE;
			errlightcontrolstate := 30;	// next state
		END_IF
	30:
		ErrLightTimer(in := TRUE, pt := ErrLightFinishTime);
		IF ErrLightTimer.Q THEN
			errlightcontrolstate := 0;
		END_IF
END_CASE

(* legacy ------
// read di
Read_6Ax_DI(Enable:=Num_of_axis_GV > 0, Offset:=143, Value=>DI_Raw);
new_DI_Value := UDINT_TO_UINT(DI_Raw);	// need convert to UINT otherwise it contain much more unwanted bits, it's not necessary but just keep this line to remember
// judge which bit is true
FOR forCounter := 1 TO UINT_TO_INT(SIZEOF(Read_DI)) DO // loop all bool value
	Read_DI[forCounter] := UINT_TO_BOOL(new_DI_Value AND SHL(1, forCounter - 1));
END_FOR

// write do
new_Do_Value:= 0;	// initialize 

(*	useless too complicated, no need to do the real calculation
FOR forCounter := 0 TO UINT_TO_INT(SIZEOF(SetDo)) DO // loop all bool value
	IF SetDo[forCounter] THEN	// if out put is true
		squareValue := 1;	// first value is 1, 2^0=1
		IF forCounter <> 0 THEN // if is not first value
			FOR squareCounter := 1 TO forCounter DO	// calculate dec value
				squareValue := squareValue * 2;
			END_FOR
		END_IF
		DoValue := DoValue + INT_TO_UINT(squareValue);
	END_IF
END_FOR
*)
// shift mamary according to bool
FOR forCounter := 1 TO UINT_TO_INT(SIZEOF(Set_Do)) DO // loop all bool value
	IF Set_Do[forCounter] THEN	// if out put is true
		new_Do_Value := new_Do_Value + SHL(1, forCounter - 1);
	END_IF
END_FOR

IF new_Do_Value <> old_Do_Value THEN
	old_Do_Value := new_Do_Value;
END_IF
Write_6Ax_Do(Enable:=Num_of_axis_GV > 0, Offset:=143, Value:=old_Do_Value);	// write DO
---------*)
// debug
IF NOT starter THEN
	starter := TRUE;
	found_0 := found_1 := found_2 := FALSE;
	offsetValue := 0;
END_IF
TestAin_0(enable:= TRUE, offset :=offsetValue, value=>read_0);
TestAin_1(enable:= TRUE, offset :=offsetValue, value=>read_1);
TestAin_2(enable:= TRUE, offset :=offsetValue, value=>read_2);

IF read_0 > try THEN
	try := read_0 - MaxmentOffset;
END_IF
try2 := (UINT_TO_REAL(read_0)/UINT_TO_REAL(try))*100;

IF read_0 > target_low AND read_0 < target_high THEN
	found_0 := TRUE;
END_IF

IF read_1 > target_low AND read_1 < target_high THEN
	found_1 := TRUE;
END_IF

IF read_2 > target_low AND read_2 < target_high THEN
	found_2 := TRUE;
END_IF

IF NOT found_0 AND NOT found_1 AND NOT found_2 OR maunl_next THEN
	offsetValue := offsetValue + 1;
	maunl_next := found_0 := found_1 := found_2 := FALSE;
END_IF

//Debug area start-------------------------------------------------------------------
// read how many axis has been config
ReadCfg(axisnumber => Num_of_axis);
FOR cfg_i := 0 TO WORD_TO_INT(Num_of_axis) - 1 DO
	PowerState[cfg_i](axis := cfg_i, enable := TRUE);
	AxisMeasure[cfg_i](axis := cfg_i, enable := TRUE);
	IF PowerState[cfg_i].State = 3 THEN // servo lost or error
		Servo_Testment_State := -40;
	END_IF
END_FOR


PowerState[0].State;
PowerState[1].State;
PowerState[2].State;
PowerState[3].State;
PowerState[4].State;
PowerState[5].State;
PowerState[0].Valid;
PowerState[1].Valid;
PowerState[2].Valid;
PowerState[3].Valid;
PowerState[4].Valid;
PowerState[5].Valid;
AxisMeasure[0].Valid;
AxisMeasure[1].Valid;
AxisMeasure[2].Valid;
AxisMeasure[3].Valid;
AxisMeasure[4].Valid;
AxisMeasure[5].Valid;
AxisMeasure[0].Pos;
AxisMeasure[1].Pos;
AxisMeasure[2].Pos;
AxisMeasure[3].Pos;
AxisMeasure[4].Pos;
AxisMeasure[5].Pos;
AxisMeasure[0].Speed;
AxisMeasure[1].Speed;
AxisMeasure[2].Speed;
AxisMeasure[3].Speed;
AxisMeasure[4].Speed;
AxisMeasure[5].Speed;
AxisMeasure[0].Torque;
AxisMeasure[1].Torque;
AxisMeasure[2].Torque;
AxisMeasure[3].Torque;
AxisMeasure[4].Torque;
AxisMeasure[5].Torque;
AxisMeasure[0].Acc;
AxisMeasure[1].Acc;
AxisMeasure[2].Acc;
AxisMeasure[3].Acc;
AxisMeasure[4].Acc;
AxisMeasure[5].Acc;

// speed control test
IF NOT sc_enb THEN
	SC_State := 0;
END_IF
CASE SC_State OF
	-10:	// error will moving
	0:
		IF SC_Enb THEN
			FOR sc_i := 0 TO 5 DO
				SpeedMovFir[sc_i](axis := sc_i,execute := FALSE);
				SpeedMovSec[sc_i](axis := sc_i,execute := FALSE);
			END_FOR
			SCTimer(in := FALSE);
			SCGroupSwitch := FALSE;
			sc_state := 10;
		END_IF
	10:
		SCTimer(in := TRUE, pt := SCMovTime);
		IF SCTimer.Q THEN	// if time reached
			IF NOT SCGroupSwitch THEN	//decide which motor group is time to switch dir
				SCGroupSwitch := TRUE;
				IF SCFirDir = mcPositiveDirection THEN	// if first group is moving positivily
					SCFirDir := mcNegativeDirection;	// then switch to negative
				ELSE
					SCFirDir := mcPositiveDirection;
				END_IF
			ELSE
				SCGroupSwitch := FALSE;
				IF SCSecDir = mcPositiveDirection THEN
					SCSecDir := mcNegativeDirection;
				ELSE
					SCSecDir := mcPositiveDirection;
				END_IF
			END_IF
		END_IF
		FOR sc_i := 0 TO 5 BY 2 DO
			SpeedMovFir[sc_i](axis := sc_i,execute := NOT (SCTimer.Q AND SCGroupSwitch)	// only switch off when timer is alarted and first group direction is switched
				, velocity := SCVel, Acceleration := SCACC, Deceleration := SCACC, Jerk := SCJerk
				, Direction := SCFirDir, Buffermode := mcAborting);
			IF SpeedMovFir[sc_i].Error THEN
				SC_State := -10;
			END_IF
		END_FOR
		FOR sc_i := 1 TO 5 BY 2 DO
			SpeedMovSec[sc_i](axis := sc_i,execute := NOT (SCTimer.Q AND NOT SCGroupSwitch)	// only switch off when timer is alarted and second group direction is switched
				, velocity := SCVel, Acceleration := SCACC, Deceleration := SCACC, Jerk := SCJerk
				, Direction := SCSecDir, Buffermode := mcAborting);
			IF SpeedMovSec[sc_i].Error THEN
				SC_State := -10;
			END_IF
		END_FOR
		
		IF SCTimer.Q THEN	// if time reached
			SCTimer(in := FALSE);	// switch off timer
		END_IF
END_CASE


//Debug area end-------------------------------------------------------------------

END_PROGRAM

// CODESYS_Control_x86_Arca_Control_SM/Application/IO_Management/Digital_Input
FUNCTION_BLOCK Digital_Input
VAR_INPUT
	enable : BOOL;
END_VAR
VAR_OUTPUT
	DI_Array : ARRAY [1..12] OF BOOL;
	DI_01 : BOOL;
	DI_02 : BOOL;
	DI_03 : BOOL;
	DI_04 : BOOL;
	DI_05 : BOOL;
	DI_06 : BOOL;
	DI_07 : BOOL;
	DI_08 : BOOL;
	DI_09 : BOOL;
	DI_10 : BOOL;
	DI_11 : BOOL;
	DI_12 : BOOL;
	DI_13 : BOOL;
	DI_14 : BOOL;
	DI_15 : BOOL;
	DI_16 : BOOL;
	DI_17 : BOOL;
	DI_18 : BOOL;
	DI_19 : BOOL;
	DI_20 : BOOL;
	DI_21 : BOOL;
	DI_22 : BOOL;
	DI_23 : BOOL;
	DI_24 : BOOL;
END_VAR
VAR
	forCounter: INT;
	
	Read_6Ax_DI: Arcalibrary.ECAT_GetPdi_U32;
	DI_Raw : UDINT;
END_VAR

// read di
Read_6Ax_DI(Enable:= enable, Offset:=143, Value=>DI_Raw);

// judge which bit is true
FOR forCounter := 1 TO UINT_TO_INT(SIZEOF(DI_Array)) DO // loop all bool value
	DI_Array[forCounter] := UDINT_TO_BOOL(DI_Raw AND SHL(1, forCounter - 1));
END_FOR

DI_01 := DI_Array[01];
DI_02 := DI_Array[02];
DI_03 := DI_Array[03];
DI_04 := DI_Array[04];
DI_05 := DI_Array[05];
DI_06 := DI_Array[06];
DI_07 := DI_Array[07];
DI_08 := DI_Array[08];
DI_09 := DI_Array[09];
DI_10 := DI_Array[10];
DI_11 := DI_Array[11];
DI_12 := DI_Array[12];
(*	// not yet ready, need add more code for second driver for more input
DI_13 := DI_Array[13];
DI_14 := DI_Array[14];
DI_15 := DI_Array[15];
DI_16 := DI_Array[16];
DI_17 := DI_Array[17];
DI_18 := DI_Array[18];
DI_19 := DI_Array[19];
DI_20 := DI_Array[20];
DI_21 := DI_Array[21];
DI_22 := DI_Array[22];
DI_23 := DI_Array[23];
DI_24 := DI_Array[24];
*)

END_FUNCTION_BLOCK

// CODESYS_Control_x86_Arca_Control_SM/Application/IO_Management/Digital_Output
FUNCTION_BLOCK Digital_Output
VAR_INPUT
	enable : BOOL;
	DO_Array: ARRAY [1..8] OF BOOL;
	DO_01 : BOOL;
	DO_02 : BOOL;
	DO_03 : BOOL;
	DO_04 : BOOL;
	DO_05 : BOOL;
	DO_06 : BOOL;
	DO_07 : BOOL;
	DO_08 : BOOL;
END_VAR
VAR_OUTPUT
END_VAR
VAR
	forCounter: INT;
	
	Set_Do: ARRAY [1..8] OF BOOL;
	new_Do_Value, old_Do_Value : UINT;
	Write_6Ax_Do: Arcalibrary.ECAT_SetPdo_U32;
END_VAR

// write do
new_Do_Value:= 0;	// initialize 
Set_Do[01] := DO_Array[01] OR do_01;
Set_Do[02] := DO_Array[02] OR do_02;
Set_Do[03] := DO_Array[03] OR do_03;
Set_Do[04] := DO_Array[04] OR do_04;
Set_Do[05] := DO_Array[05] OR do_05;
Set_Do[06] := DO_Array[06] OR do_06;
Set_Do[07] := DO_Array[07] OR do_07;
Set_Do[08] := DO_Array[08] OR do_08;

// shift mamary according to bool
FOR forCounter := 1 TO UINT_TO_INT(SIZEOF(Set_Do)) DO // loop all bool value
	IF DO_Array[forCounter] THEN	// if out put is true
		new_Do_Value := new_Do_Value + SHL(1, forCounter - 1);
	END_IF
END_FOR

IF new_Do_Value <> old_Do_Value THEN
	old_Do_Value := new_Do_Value;
END_IF
Write_6Ax_Do(Enable:= enable, Offset:=143, Value:=old_Do_Value);	// write DO

END_FUNCTION_BLOCK

// CODESYS_Control_x86_Arca_Control_SM/Application/IO_Management/Digital_Input_Analog
FUNCTION_BLOCK Digital_Input_Analog
VAR_INPUT
	enable : BOOL;
	MaxRawInputValue : ARRAY[0..7] OF UINT;
	MinRawInputValue :  ARRAY[0..7] OF UINT;
	MaxmentOffset : UINT := 50;
	SmoothTIme : TIME := T#200MS;
END_VAR
VAR_OUTPUT
	DIA_raw: ARRAY[0..7] OF UINT;
	DIA_Process : ARRAY[0..7] OF REAL;
END_VAR
VAR
	_Timer : ton;
	_sample_times : UINT;
	
	_DA: Arcalibrary.ECAT_GetPdi_U16;
	_offset : ARRAY[0..7] OF WORD;
	_raw_value : ARRAY[0..7] OF UDINT;
END_VAR

_offset[0]:=147;
_DA(enable:= enable, offset := _offset[0]);

_Timer(in:= TRUE, pt := SmoothTime);
_raw_value[0] := _raw_value[0] + _DA.Value;
_sample_times := _sample_times + 1;
IF _Timer.Q THEN
	DIA_raw[0] := UDINT_TO_UINT(_raw_value[0] / UINT_TO_UDINT(_sample_times));
	_raw_value[0] := 0;
	_sample_times := 0;
	_Timer (in := FALSE);
END_IF

DIA_Process[0] := (UINT_TO_REAL(DIA_raw[0])/UINT_TO_REAL((MaxRawInputValue[0] - MinRawInputValue[0]) - MaxmentOffset))*100;

IF DIA_Process[0] > 100 THEN
	DIA_Process[0] := 100;
END_IF

IF DIA_Process[0] < 0 THEN
	DIA_Process[0] := 0;
END_IF

END_FUNCTION_BLOCK

// CODESYS_Control_x86_Arca_Control_SM/Application/Testment_Servo_Function_Test/Testment_Message_Manager
FUNCTION_BLOCK Testment_Message_Manager
VAR_INPUT
	state_in : INT;
END_VAR
VAR_OUTPUT
	Start_Restart_indicator : BOOL;
	Show_Message : WSTRING;
	Error_State : BOOL;
END_VAR
VAR
	_case : int;
END_VAR

_case := state_in;

IF state_in < 0 THEN
	Error_State := TRUE;
ELSE 
	Error_State := FALSE;
END_IF

IF state_in <> 0 THEN
	Start_Restart_indicator := FALSE;
END_IF

CASE _case OF 
	-50:
		Show_Message := " 错误_50 ";
	-45:
		Show_Message := " 错误_45 ";
	-40:
		Show_Message := " 错误_40 ";
	-35:
		Show_Message := " 错误_35 ";
	-33:
		Show_Message := " 错误_33 ";
	-30:
		Show_Message := " 错误_30 ";
	-20:
		Show_Message := " 错误_20 ";
	-10:
		Show_Message := " 错误_10 ";
	-5:
		Show_Message := " 错误_5 ";
	0:
		Start_Restart_indicator := TRUE;
		Show_Message := " 步骤_0 ";
	20:
		Show_Message := " 步骤_20 ";
	50:
		Show_Message := " 步骤_50 ";
	100:
		Show_Message := " 步骤_100 ";
	110:
		Show_Message := " 步骤_110 ";
	130:
		Show_Message := " 步骤_130 ";
	
	//140:	
	//	Show_Message := " 完成 ";
	
END_CASE

END_FUNCTION_BLOCK

// CODESYS_Control_x86_Arca_Control_SM/Application/AxisControl/MultiAxisABSMove
FUNCTION_BLOCK MultiAxisABSMove
VAR_INPUT
	FirstAuxAxisNum : BYTE;	// for safty reason, this block do not accept different axis after enabled
	LastAuxAxisNum : BYTE;
	Enable : BOOL;
	Axis_Mov_Indicator : ARRAY [0..255] OF BOOL; // tell program which axis to mov whih not mov
	Axis_Mov_Pos : ARRAY [0..255] OF REAL; // tell program which axis to what position
	Execute : BOOL;
	Vel, Acc, Dec, Jerk : REAL;	// not allow 0 or none input
	MoveMethod : MutiAxisMoveMethod;
END_VAR
VAR_OUTPUT
	done : BOOL;
	error : BOOL;
	error_str : STRING;
END_VAR
VAR
	_Faxis, _Laxis : BYTE;	// internal first axis and last axis
	_Indicator : ARRAY [0..255] OF BOOL; // internal indicator
	_enb : BOOL;
	_state : INT;
	_axisMovCmd : ARRAY [0..255] OF ArcaLibrary.MC_MoveAbsolute;
	_i : INT;
	_totalMovAxis : WORD;
	_totalMovDone : WORD;
	_err_axis : INT;
	_err_header : STRING := 'Error State: ';
	_pos : ARRAY [0..255] OF REAL;
	_speedPar : ARRAY [0..255] OF ARRAY [0..3] OF REAL;	// 255 velocity, acceleration, deceleration and jerk
	_maxDistance, _maxArriveTime : REAL;
	_readPos : ARRAY [0..255] OF ArcaLibrary.MCAT_ReadAxisMeasures;
	_currPos : ARRAY [0..255] OF REAL;
	_accRatio, _decRatio, _jerkRatio : REAL;
END_VAR


IF NOT enable THEN
	IF _enb THEN	// if local enable is turn on reset values
		FOR _i := _Faxis TO _Laxis DO	// reset all cmd block
			_axisMovCmd[_i](axis :=_i, execute := FALSE);
			_readPos[_i](axis := _i, enable := FALSE);
		END_FOR
		_enb :=
		done :=
		error := FALSE;
		delete(error_str, len := UINT_TO_INT(SIZEOF(error_str)), pos := 1);
		_state := 0;
	END_IF
	RETURN;
END_IF
IF NOT _enb THEN	// initialze
	_enb := TRUE;
	_Faxis := FirstAuxAxisNum;	// for safty reason, this block do not accept different axis after enabled
	_Laxis := LastAuxAxisNum;
	FOR _i := _Faxis TO _Laxis DO	// reset all cmd block
		_axisMovCmd[_i](axis :=_i, execute := FALSE);
	END_FOR
END_IF

CASE _state OF
	-10:
		error := TRUE;
		error_str := concat(_err_header,concat(INT_TO_STRING(_state), concat( ', Axis move block error. Error axis number is: ', INT_TO_STRING(_err_axis))));
	-2:
		error := TRUE;
		error_str := concat(_err_header,concat(INT_TO_STRING(_state), ', speed parameter input is 0'));
	-1:
		error := TRUE;
		error_str := concat(_err_header,concat(INT_TO_STRING(_state), ', there are no such MoveMethod as given'));
	0:
		IF execute THEN
			IF vel = 0 OR acc = 0 OR dec = 0 OR jerk = 0 THEN
				_state := -2;
				RETURN;
			END_IF
			_pos := Axis_Mov_Pos;	// transfer to local value for safe
			_Indicator := Axis_Mov_Indicator;
			CASE MoveMethod OF
				0:	
					FOR _i := _Faxis TO _Laxis DO
						_speedPar[_i][0] := vel;
						_speedPar[_i][1] := acc;
						_speedPar[_i][2] := dec;
						_speedPar[_i][3] := jerk;
					END_FOR
				10:	// calculate all axis insure them arrive destination
					_accRatio := acc/vel;	// accRaito
					_decRatio := dec/vel;	// decRaito
					_jerkRatio := jerk/acc;	// JerkaRito
					FOR _i := _Faxis TO _Laxis DO	// find which axis have most far destination
						IF _Indicator[_i] THEN
							_readPos[_i](axis := _i, enable := TRUE, pos => _currPos[_i]);
							IF _maxDistance < ABS(_currPos[_i] - _pos[_i]) THEN
								_maxDistance := ABS(_currPos[_i] - _pos[_i]);
							END_IF
							_readPos[_i](axis := _i, enable := FALSE);
						END_IF
					END_FOR
					_maxArriveTime := _maxDistance/vel;
					FOR _i := _Faxis TO _Laxis DO	// calculate individual speed parameter for each axis
						IF _Indicator[_i] THEN
							_speedPar[_i][0] := ABS(_currPos[_i] - _pos[_i])/_maxArriveTime;
							_speedPar[_i][1] := _speedPar[_i][0] * _accRatio;
							_speedPar[_i][2] := _speedPar[_i][0] * _decRatio;
							_speedPar[_i][3] := _speedPar[_i][1] * _jerkRatio;
						END_IF
					END_FOR
			ELSE
				error := TRUE;
				_state := -1;
				RETURN;
			END_CASE
			_state := 10;
		END_IF
	10:
		_totalMovAxis := _totalMovDone := 0;
		_i := _Faxis;
		
		WHILE _i <= _Laxis AND NOT error DO
			IF _Indicator[_i] THEN	// if indicator show _i motor need to be command
				_axisMovCmd[_i](axis := _i, execute := TRUE, Position := _pos[_i]
					, velocity := _speedPar[_i][0], acceleration := _speedPar[_i][1], Deceleration := _speedPar[_i][2], Jerk := _speedPar[_i][3]
					, Direction := mcShortestway, Buffermode := mcAborting);
				_totalMovAxis := _totalMovAxis + 1;	// count how many axis are indicate to move
				IF _axisMovCmd[_i].Done THEN
					_totalMovDone := _totalMovDone + 1;
				END_IF
				IF _axisMovCmd[_i].Error THEN
					error := TRUE;
					_err_axis := _i;
				END_IF
			END_IF
			_i := _i + 1;
		END_WHILE
		IF error THEN
			_state := -10;
		ELSIF NOT error AND _totalMovAxis = _totalMovDone THEN	// all axis move done and no error
			FOR _i := _Faxis TO _Laxis DO	// reset all cmd block
				_axisMovCmd[_i](axis :=_i, execute := FALSE);
			END_FOR
			done := TRUE;
			_state := 20;
		END_IF
	20:
		IF NOT execute THEN
			done := FALSE;
			_state := 0;
		END_IF
END_CASE

// debug

_axisMovCmd[00].Done;
_axisMovCmd[01].Done;
_axisMovCmd[02].Done;
_axisMovCmd[03].Done;
_axisMovCmd[04].Done;
_axisMovCmd[05].Done;
_axisMovCmd[06].Done;
_axisMovCmd[07].Done;
_axisMovCmd[08].Done;
_axisMovCmd[09].Done;
_axisMovCmd[10].Done;
_axisMovCmd[11].Done;
_axisMovCmd[12].Done;
_axisMovCmd[13].Done;
_axisMovCmd[14].Done;
_axisMovCmd[15].Done;
_axisMovCmd[16].Done;
_axisMovCmd[17].Done;

END_FUNCTION_BLOCK

// CODESYS_Control_x86_Arca_Control_SM/Application/AxisControl/MultiAxisTorqueLimit
FUNCTION_BLOCK MultiAxisTorqueLimit
VAR_INPUT
	FirstAuxAxisNum : BYTE;	// for safty reason, this block do not accept different axis after enabled
	LastAuxAxisNum : BYTE;
	Enable : BOOL;
	Axis_Torque_Limit_Indicator : ARRAY [0..255] OF BOOL; // tell program which axis to limit Torque
	Axis_Torque_Limit_Value : ARRAY [0..255] OF REAL; // tell program which axis's torque limition
	Execute : BOOL;
END_VAR
VAR_OUTPUT
	done : BOOL;
	error : BOOL;
	error_str : STRING;
END_VAR
VAR
	_Faxis, _Laxis : BYTE;	// internal first axis and last axis
	_indicator : ARRAY [0..255] OF BOOL; // internal torque indicator
	_enb : BOOL;
	_state : INT;
	_axisLimitionCmd : ARRAY [0..255] OF ArcaLibrary.MCAT_AxisSetLimits;
	_i : INT;
	_totalNeedSetAxis : WORD;
	_totalSetDone : WORD;
	_err_axis : INT;
	_err_header : STRING := 'Error State: ';

	_toque_limit : ARRAY [0..255] OF REAL;
	
END_VAR


IF NOT enable THEN
	IF _enb THEN	// if local enable is turn on reset values
		FOR _i := _Faxis TO _Laxis DO	// reset all cmd block
			_axisLimitionCmd[_i](axis :=_i, execute := FALSE);
		END_FOR
		_enb :=
		done :=
		error := FALSE;
		delete(error_str, len := UINT_TO_INT(SIZEOF(error_str)), pos := 1);
		_state := 0;
	END_IF
	RETURN;
END_IF
IF NOT _enb THEN	// initialze
	_enb := TRUE;
	_Faxis := FirstAuxAxisNum;	// for safty reason, this block do not accept different axis after enabled
	_Laxis := LastAuxAxisNum;
	FOR _i := _Faxis TO _Laxis DO	// reset all cmd block
		_axisLimitionCmd[_i](axis :=_i, execute := FALSE);
	END_FOR
END_IF

CASE _state OF
	-10:
		error := TRUE;
		error_str := concat(_err_header,concat(INT_TO_STRING(_state), concat( ', Axis move block error. Error axis number is: ', INT_TO_STRING(_err_axis))));
	-1:
		error := TRUE;
		error_str := concat(_err_header,concat(INT_TO_STRING(_state), ', there are no such MoveMethod as given'));
	0:
		IF execute THEN
			_toque_limit := Axis_Torque_Limit_Value;	// transfer to local value for safe
			_indicator := Axis_Torque_Limit_Indicator;
			_state := 10;
		END_IF
	10:
		_totalSetDone := _totalNeedSetAxis := 0;
		_i := _Faxis;
		
		WHILE _i <= _Laxis AND NOT error DO
			IF _indicator[_i] THEN	// if indicator show _i motor need to be command
				_axisLimitionCmd[_i](axis := _i, execute := TRUE, TorqueLimit := _toque_limit[_i]);
				_totalNeedSetAxis := _totalNeedSetAxis + 1;	// count how many axis are indicate to move
				IF _axisLimitionCmd[_i].Done THEN
					_totalSetDone := _totalSetDone + 1;
				END_IF
				IF _axisLimitionCmd[_i].Error THEN
					error := TRUE;
					_err_axis := _i;
				END_IF
			END_IF
			_i := _i + 1;
		END_WHILE
		IF error THEN
			_state := -10;
		ELSIF NOT error AND _totalNeedSetAxis = _totalSetDone THEN	// all axis move done and no error
			FOR _i := _Faxis TO _Laxis DO	// reset all cmd block
				_axisLimitionCmd[_i](axis :=_i, execute := FALSE);
			END_FOR
			done := TRUE;
			_state := 20;
		END_IF
	20:
		IF NOT execute THEN
			done := FALSE;
			_state := 0;
		END_IF
END_CASE

END_FUNCTION_BLOCK

// CODESYS_Control_x86_Arca_Control_SM/Application/Hand_Control_blocks/Grab_Control
FUNCTION_BLOCK Grab_Control
VAR_INPUT
	Enable : BOOL;
	OverFeed : INT;
	Grab : Grab_Command;
END_VAR
VAR_OUTPUT
	Done : BOOL;
	isMoving : BOOL;
	Error : BOOL;
	Err_Message : Error_Message;
END_VAR
VAR
	state : INT := 0;
	i : INT;
	//movment settings
	Finger_Movement: ArcaLibrary.MCAT_MoveDirectAbsolute;
	
	ReadCurrentPos : ArcaLibrary.MC_GroupReadActualPosition;
	CurrPos : ARRAY [1..6] OF REAL;
	CoordSys1: ArcaLibrary.MC_COORD_SYSTEM := mcMCS;
	
	Set1: ArcaLibrary.MCAT_Settings;
	ToolMoveVel:REAL:=100;
	ToolMoveAcc:REAL:=500;
	ToolMoveJrk:REAL:=2500;
	bufmode: ArcaLibrary.MC_BUFFER_MODE:=mcBuffered;
	transition: ArcaLibrary.MC_TRANSITION_MODE:=tmRelativeCornerDistance;
	tmPar: ARRAY [1..12] OF REAL :=[1.0, 1.0, 1.0, 1.0, 1.0, 1.0, 1.0, 1.0, 1.0, 1.0, 1.0, 1.0];

	Pos_For_Hand_Block : ArcaLibrary.MCAT_Position;
	Position_0: ARRAY [1..6] OF REAL :=[0.300, -0.100, 0.200, 160.0, 180.0, 0.0];
	Position_1: ARRAY [1..6] OF REAL :=[0.500, -0.100, 0.200, 160.0, 180.0, 0.0];
	RobotMovPos: ARRAY [1..6] OF REAL :=[0.50, -0.100, 0.200, 160.0, 180.0, 0.0];
	
	AxesPosForExternal: ARRAY [1..32] OF REAL;
	
	MaxDifference : REAL := 0.005;
	
	// grab pos
	g_grab: ARRAY [1..32] OF REAL;
	
	// max degree for every motor
	Root_min : REAL := 235;
	Root_max : REAL := 350;
	
	Tip_min : REAL := 140;
	Tip_max : REAL := 40;
	
	
	grab_angle_min : REAL := 0;
	grab_angle_max : REAL := 180;
	
	// debug
	mid_0_max: REAL;
	mid_0_min: REAL;
	
	clamp : Value_Clamp;
END_VAR

IF NOT Enable AND state > 0 THEN
	state := 0;
END_IF

IF overfeed > 90 THEN
	overfeed := 90;
ELSIF overfeed < 0 THEN
	overfeed := 0;
END_IF

// read current virtual robot postion
ReadCurrentPos(axesGroup := 0, execute := state > 0, CoordSystem:=mcMcs, Position=>CurrPos);
IF ReadCurrentPos.Error THEN
	state := -10;
END_IF

CASE state OF
	-30:
		error := TRUE;
		Err_Message := error_message.Err_AuxAxis_Movement_Block_err;
	-10:
	(*
		IF ReadCurrentPos.ErrorID THEN
			
		END_IF
	*)
		error := TRUE;
		Err_Message := error_message.Err_AuxAxis_Movement_Cannot_read_virture_robot_position;
		
	0:
		Done := error := FALSE;
		Err_Message := error_message.Err_None;
		
		IF Enable THEN
			state := 10;
		END_IF

	10:	//initialize
	
		// set position
		// clamp Root_Angle
		clamp(current := Grab.Root_Angle, first_value := Root_min, second_value := Root_max, newV => g_grab[1]);
		
		// clamp Tip_Angle
		clamp(current := Grab.Tip_Angle, first_value := Tip_min, second_value := Tip_max, newV => g_grab[2]);
		
		// clamp Tip_Angle
		clamp(current := Grab.Clamp_Angle, first_value := grab_angle_min, second_value := grab_angle_max, newV => g_grab[3]);
		
		// take a judge to find where is the robot and give a different destination
		IF ABS(CurrPos[1] - Position_0[1]) > MaxDifference THEN
			RobotMovPos := Position_0;
		ELSE 
			RobotMovPos := Position_1;
		END_IF
		
		// asign value for hand movment block
		Pos_For_Hand_Block.Position := RobotMovPos;
		Pos_For_Hand_Block.AxesPosition:=AxesPosForExternal;
		Pos_For_Hand_Block.AuxAxes:=g_grab;
		Pos_For_Hand_Block.CoordSystem:=CoordSys1;
		
		Set1.Velocity:=ToolMoveVel;
		Set1.Acceleration:=ToolMoveAcc;
		Set1.Deceleration:=ToolMoveAcc;
		Set1.Jerk:=ToolMoveJrk;
		Set1.OverfeedPerc:=Overfeed;
		Set1.BufferMode:=bufmode;
		Set1.TransitionMode:=transition;
		Set1.TransitionParameter:=tmPar;
		
		Finger_Movement(AxesGroup:=0, Execute:=FALSE);
		State := 20;
	20:
		IF (NOT enable) THEN
			State := 0;
		END_IF
		
		Finger_Movement(AxesGroup:=0, Execute:=TRUE, Position:=Pos_For_Hand_Block, Settings:=Set1, active => isMoving);
		
		IF Finger_Movement.Done THEN
			Finger_Movement(AxesGroup:=0, Execute:=FALSE);
			state := 50;
		ELSIF Finger_Movement.Error OR Finger_Movement.CommandAborted THEN
			state := -30;
		END_IF
	50:
		done := TRUE;
END_CASE
// end of the program

END_FUNCTION_BLOCK

// CODESYS_Control_x86_Arca_Control_SM/Application/Utility_functions/Value_Clamp
FUNCTION_BLOCK Value_Clamp
// clamp the input value between first value and second value
VAR_INPUT
	Current : REAL;
	First_Value : REAL;
	Second_value : REAL;
END_VAR
VAR_OUTPUT
	newV : REAL;
END_VAR
VAR
END_VAR

newV := Current;
IF First_Value < Second_value THEN
	IF Current < First_Value THEN
		newV := First_Value;
	END_IF
	IF Current > Second_value THEN
		newV := Second_value;
	END_IF
ELSIF First_Value > Second_value THEN
	IF Current > First_Value THEN
		newV := First_Value;
	END_IF
	IF Current < Second_value THEN
		newV := Second_value;
	END_IF
END_IF
// not going to deal the situation of first value equal to second value

END_FUNCTION_BLOCK

// CODESYS_Control_x86_Arca_Control_SM/Application/Hand_Control_blocks/Grab_Demo
FUNCTION_BLOCK Grab_Demo
VAR_INPUT
	enable :BOOL;
	internal_hand_enable : BOOL;
	startMov :BOOL;
	ovr : INT;
END_VAR

VAR_OUTPUT
	IsEnabled : BOOL;
	IsMoving : BOOL;
	err : BOOL;
	err_message : error_message;
END_VAR

VAR
	// state control
	cycleState : INT;	// state machine
	cycleCounter : INT;	// counte how many time already been done
	start_cycle : INT := 1;	// start cycle from a number
	total_cycle_time : INT := 24; //	max cycle time
	cycleTimer : ton;
	cycleDelayTime : TIME := T#500MS;	// delay time between every gesture
	
	// hand powerOn
	powerHand : BOOL;
	powerOnHand : AuxAxis_PowerOn;
	_enabled : BOOL;
	
	// gestrure mov block
	GrabMov : Grab_Control;
	GrabCmd : grab_command;
	_GrabCmdEmpt : grab_command;
END_VAR


//err
IF powerOnHand.Error OR GrabMov.Error THEN
	err := TRUE;
	IF powerOnHand.Error THEN
		err_message := powerOnHand.Err_Message;
	ELSIF GrabMov.Error THEN
		err_message := GrabMov.Err_Message;
	END_IF
ELSE
	err := FALSE;
	err_message := error_message.Err_None;
END_IF

// enable hand
IF internal_hand_enable THEN
	powerOnHand(enable := enable);
	_enabled := IsEnabled := powerOnHand.Done;
END_IF

IF NOT enable THEN
	cycleState := 0;
	isMoving := FALSE;
	cycleTimer(in := FALSE);	// reset timer
	GrabMov(Enable := FALSE);	// reset movement block
END_IF

CASE cycleState OF
	0: 
		// if block is enabled and order to move and (manager by internal power or by external power)
		IF enable AND startMov AND (NOT internal_hand_enable OR _enabled) THEN
			GrabCmd.Root_Angle := 200;	// all open
			GrabCmd.Tip_Angle := 200;
			GrabCmd.Clamp_Angle := 0;
			
			cycleCounter := start_cycle;	// set counter to start_cycle
			cycleState := 10;
		END_IF
	10:
		GrabMov(Enable := TRUE, overfeed := ovr,Grab := GrabCmd, isMoving => isMoving);
		IF GrabMov.Done THEN
			cycleTimer(in := TRUE, pt:= cycleDelayTime);	// start timer for delay
			IF cycleTimer.Q THEN	// time reach
				cycleCounter := cycleCounter + 1;	// done and self add for next gesture
				cycleTimer(in := FALSE);	// reset timer
				GrabMov(Enable := FALSE);	// reset movement block
				
				IF cycleCounter <= total_cycle_time THEN
					IF cycleCounter <= 5 THEN	// first movement, root as clamp
						IF GrabCmd.Root_Angle <> 400 THEN // if not clamp
							GrabCmd.Root_Angle := 400;	// root in max
							GrabCmd.Tip_Angle := 90;	// tip mov in middle
						ELSE
							GrabCmd.Root_Angle := 200;	// root in open
							GrabCmd.Tip_Angle := 200;	// tip in open
						END_IF
					ELSIF cycleCounter <= 9 THEN	// second movement, show tip movement
						IF GrabCmd.Tip_Angle <> 40 THEN // if not clmap
							GrabCmd.Root_Angle := 200;	// root in open
							GrabCmd.Tip_Angle := 40;	// tip max
						ELSE
							GrabCmd.Root_Angle := 200;	// root in open
							GrabCmd.Tip_Angle := 200;	// tip in open
						END_IF
					ELSIF cyclecounter <= 15 THEN	// second movement, tip as clamp
						IF GrabCmd.Tip_Angle <> 40 THEN
							GrabCmd.Root_Angle := 300;	// root mov to mid
							GrabCmd.Tip_Angle := 40;	// tip max
						ELSE
							GrabCmd.Root_Angle := 200;	// root in open
							GrabCmd.Tip_Angle := 140;	// tip in open
						END_IF
					ELSIF cyclecounter <= 18 THEN	// third movement, show clamp angle
						IF GrabCmd.Clamp_Angle <> 180 THEN
							GrabCmd.Clamp_Angle := 180;	// clamp angle to max
						ELSE
							GrabCmd.Clamp_Angle := 0;	// clamp angle to min
						END_IF
					ELSIF cyclecounter <= 24 THEN	// fouth movement, tip as clamp in another clamp angle
						IF GrabCmd.Tip_Angle <> 40 THEN
							GrabCmd.Root_Angle := 300;	// root mov to mid
							GrabCmd.Tip_Angle := 40;	// tip max
						ELSE
							GrabCmd.Root_Angle := 200;	// root in open
							GrabCmd.Tip_Angle := 140;	// tip in open
						END_IF
					END_IF
					cycleState := 10;	// if not reach total number then go back keep do next gesture
				ELSE
					cycleState := 0;	// if reach maximum then go back beginning
				END_IF
			END_IF
		END_IF
END_CASE

END_FUNCTION_BLOCK

// CODESYS_Control_x86_Arca_Control_SM/Application/Hand_Control_blocks/Hand_Gesture
FUNCTION_BLOCK Hand_Gesture
VAR_INPUT
	Enable : BOOL;
	OverFeed : INT;
	Gesture : Gesture_Type;
	HandType : PhysicalHandType;
	HandFirstAxis : BYTE;
	HandLastAxis : BYTE;
	HandAxisAllowToMov : ARRAY [0..17] OF BOOL;
END_VAR
VAR_OUTPUT
	Done : BOOL;
	isMoving : BOOL;
	Error : BOOL;
	Err_Message : Error_Message;
END_VAR
VAR
	_enb : BOOL;
	state : INT := 0;
	i : INT;
	//movment settings
	_ov : REAL;
	FingerMovPos: ARRAY [1..32] OF REAL;
	SecFingerMovPos: ARRAY [1..32] OF REAL;
	ThdFingerMovPos: ARRAY [1..32] OF REAL;
	CycleMovTimes : INT := 1;
	CycleMovDone : BOOL;
	
	CycleFingerMovPos: ARRAY [0..20] OF ARRAY[1..32] OF REAL;	
	DelayTimer : ton;
	DelayTime : ARRAY [0..20] OF TIME;
	readyToMov : BOOL;
	G_MovObj_Muilt : INT;
	
	MultisingleMov : MultiAxisABSMove;
	MultiMov_for_counter : INT;
	Give_Finger_Pos_Counter : INT;
	GivHandPos : ARRAY [0..255] OF REAL;
	handVel : REAL := 402;	// 402 = 67rpm
	handAcc : REAL := 4020;
	handJerk : REAL := 40200;
	givenVel, givenAcc, givenJerk : REAL;
	ArrayTotalNum : INT;
	ArrayFirstRow : INT;
	ReadTorque : ARRAY [0..255] OF ArcaLibrary.MCAT_ReadAxisMeasures;
	ReadTorque_For : INT;
	HandAxisTorqueValue_Sum : ARRAY [0..255] OF REAL;
	HandAxisTorqueValue_Raw : ARRAY [0..255] OF REAL;
	HandAxisTorqueValue_Smooth: ARRAY [0..255] OF REAL;
	TorqueSmoothTime : TIME := T#2S;
	TorqueSmoothTimer : ton;
	TorqueSmoothLoopTime : BYTE;
	// gesture pos
	g_RestPos: ARRAY [1..32] OF REAL;
	g_one: ARRAY [1..32] OF REAL;
	g_two: ARRAY [1..32] OF REAL;
	g_three: ARRAY [1..32] OF REAL;
	g_four: ARRAY [1..32] OF REAL;
	g_five: ARRAY [1..32] OF REAL;
	g_six: ARRAY [1..32] OF REAL;
	g_plam: ARRAY [1..32] OF REAL;
	g_fist: ARRAY [1..32] OF REAL;
	g_thumbUp: ARRAY [1..32] OF REAL;
	
	// max degree for every motor
	wrist_0_min : REAL := 0;
	wrist_0_max : REAL := 58;
	wrist_1_min : REAL := 0;
	wrist_1_max : REAL := 58;
	
	// axis 0 to axis 2
	thumb_group_pos_0 : ARRAY[0..2] OF REAL := [000, 005, 002];		// thump relex and thump tip open
	thumb_group_pos_1 : ARRAY[0..2] OF REAL := [000, 078, 002];		// thump relex and thump tip close	// this has been used in gesture fingerwave
	thumb_group_pos_2 : ARRAY[0..2] OF REAL := [120, 005, 073];		// thumb close and thump tip open	// this has been assigned to most case when thumb need to close
	thumb_group_pos_3 : ARRAY[0..2] OF REAL := [120, 078, 073];		// thumb close and thump tip close
	thumb_3_min : REAL := 0;
	thumb_3_max : REAL := 5;
	(*
	thumb_0_min : REAL := 0;
	thumb_0_max : REAL := 120;
	thumb_1_min : REAL := 5;
	thumb_1_max : REAL := 78;
	thumb_2_min : REAL := 2;
	thumb_2_max : REAL := 73;
	*)
	
	index_0_min : REAL := 0;
	index_0_max : REAL := 20;
	index_1_min : REAL := 2;
	index_1_max : REAL := 74;
	index_2_min : REAL := 1;
	index_2_max : REAL := 87;
		
	mid_0_min : REAL := 0;
	mid_0_max : REAL := 15;
	mid_1_min : REAL := 3;
	mid_1_max : REAL := 66;
	mid_2_min : REAL := 2;
	mid_2_max : REAL := 68;
			
	ring_0_min : REAL := 0;
	ring_0_max : REAL := 10;
	ring_1_min : REAL := 2;
	ring_1_max : REAL := 53;
	ring_2_min : REAL := 2;
	ring_2_max : REAL := 68;
		
	little_0_min : REAL :=0;
	little_0_max : REAL := 20;
	little_1_min : REAL := 3;
	little_1_max : REAL := 81;
	little_2_min : REAL := 1;
	little_2_max : REAL := 78;
	
	// debug
	//temp_HandType : PhysicalHandType := motor18;
	AxisAllowToMov : ARRAY [0..255] OF BOOL;
	faxis: BYTE;	// first finge axis number
	laxis : BYTE;	// last finger axis number
END_VAR

IF NOT Enable THEN
	IF _enb THEN
		_enb := done := error := FALSE;
		Err_Message := error_message.Err_None;
		state := 0;
		MultisingleMov (enable := FALSE);
		FOR readtorque_for := faxis TO laxis DO
			ReadTorque[readtorque_for](Axis := readtorque_for, Enable := FALSE);
		END_FOR
	END_IF
	RETURN;
END_IF
IF NOT _enb THEN
	_enb := TRUE;
	faxis := HandFirstAxis;	// give initialize value from globe value
	laxis := HandLastAxis;
	FOR MultiMov_for_counter := faxis TO laxis DO
		AxisAllowToMov[MultiMov_for_counter] := HandAxisAllowToMov[MultiMov_for_counter - faxis];
	END_FOR
	TorqueSmoothTimer(in := FALSE);
END_IF

_ov := overfeed;
IF _ov > 100 THEN
	_ov := 100;
ELSIF _ov < 1 THEN
	_ov := 1;
END_IF

givenVel := handVel * (_ov/100.0);
givenAcc := handAcc * (_ov/100.0);
givenJerk := handJerk * (_ov/100.0);

// read hand axis torque and smooth in time
TorqueSmoothTimer(in := TRUE, pt := TorqueSmoothTime);
IF TorqueSmoothTimer.Q THEN
	FOR readtorque_for := faxis TO laxis DO
		IF AxisAllowToMov[readtorque_for] THEN
			HandAxisTorqueValue_Smooth[readtorque_for] 
				:= HandAxisTorqueValue_Sum [readtorque_for] / TorqueSmoothLoopTime;
			HandAxisTorqueValue_Sum[readtorque_for] := 0;
		END_IF
	END_FOR
	TorqueSmoothLoopTime := 0;
	TorqueSmoothTimer(in := FALSE);
END_IF

FOR readtorque_for := faxis TO laxis DO	// read current torque
	IF AxisAllowToMov[readtorque_for] THEN
		ReadTorque[readtorque_for](Axis := readtorque_for, Enable := TRUE
			, Torque => HandAxisTorqueValue_Raw [readtorque_for]);
		HandAxisTorqueValue_Sum[readtorque_for] 
			:= HandAxisTorqueValue_Sum[readtorque_for] + HandAxisTorqueValue_Raw [readtorque_for];
	END_IF
END_FOR
TorqueSmoothLoopTime := TorqueSmoothLoopTime + 1;

MultisingleMov(firstAuxAxisNum := faxis, LastAuxAxisNum := laxis, enable := Enable);
CASE state OF
	-50:
		error := TRUE;
	-40:
		error := TRUE;
		Err_Message := error_message.Err_Gesture_Type_Cycle_mov_block_err;
	-30:
		error := TRUE;
		Err_Message := error_message.Err_AuxAxis_Movement_Block_err;
	-20:
		error := TRUE;
		Err_Message := error_message.Err_Gesture_Type_Hand_Pos_Not_Given;
	-10:
	(*
		IF ReadCurrentPos.ErrorID THEN
			
		END_IF
	*)
		error := TRUE;
		Err_Message := error_message.Err_AuxAxis_Movement_Cannot_read_virture_robot_position;
		
	0:
		IF Enable THEN
			IF Gesture <> Gesture_Type.Gesture_Type_none THEN
				state := 10;
			ELSE 
				state := -20;
			END_IF
		END_IF

	10:	//initialize
	
		// set hand pos to relax position
		g_RestPos[01] := thumb_group_pos_0[0];	//thumb_0_min;
		g_RestPos[02] := thumb_group_pos_0[1];	//thumb_1_min;
		g_RestPos[03] := thumb_group_pos_0[2];	//thumb_2_min;
		g_RestPos[04] := thumb_3_min;
		g_RestPos[05] := index_0_min;
		g_RestPos[06] := (index_1_max - index_1_min)/2 + index_1_min;
		g_RestPos[07] := (index_2_max - index_2_min)/2 + index_2_min;
		g_RestPos[08] := mid_0_min;
		g_RestPos[09] := (mid_1_max - mid_1_min)/2 + mid_1_min;
		g_RestPos[10] := (mid_2_max - mid_2_min)/2 + mid_2_min;
		g_RestPos[11] := ring_0_min;
		g_RestPos[12] := (ring_1_max - ring_1_min)/2 + ring_1_min;
		g_RestPos[13] := (ring_2_max - ring_2_min)/2 + ring_2_min;
		g_RestPos[14] := little_0_min;
		g_RestPos[15] := (little_1_max - little_1_min)/2 + little_1_min;
		g_RestPos[16] := (little_2_max - little_2_min)/2 + little_2_min;
		g_RestPos[17] := wrist_0_min;
		g_RestPos[18] := wrist_1_min;
		
		
		//one
		g_one[01]		:= thumb_group_pos_2[0];	//thumb_0_max;		//	thumb 0
		g_one[02]		:= thumb_group_pos_2[1];	//thumb_1_max;		//	thumb 1
		g_one[03]		:= thumb_group_pos_2[2];	//thumb_2_max;		//	thumb 2
		g_one[04] 		:= thumb_3_max;
		g_one[05] 		:= g_RestPos[05];	//	index 0
		g_one[06]		:= index_1_min;		//	index 1
		g_one[07]		:= index_2_min;		//	index 2
		g_one[08] 		:= g_RestPos[08];	//	mid 0
		g_one[09]		:= mid_1_max;		//	mid 1
		g_one[10]		:= mid_2_max;		//	mid 2
		g_one[11] 		:= g_RestPos[11];	//	ring 0
		g_one[12]		:= ring_1_max;		//	ring 1
		g_one[13]		:= ring_2_max;		//	ring 2
		g_one[14] 		:= g_RestPos[14];	//	little 0
		g_one[15]		:= little_1_max;	//	little 1
		g_one[16]		:= little_2_max;	//	little 2
		g_one[17]		:= g_RestPos[17];	// wrist 0
		g_one[18]		:= g_RestPos[18];	// wrist 1
		
		
		// two
		g_two[01]		:= thumb_group_pos_2[0];	//thumb_0_max;	//	thumb 0
		g_two[02]		:= thumb_group_pos_2[1];	//thumb_1_max;	//	thumb 1
		g_two[03]		:= thumb_group_pos_2[2];	//thumb_2_max;	//	thumb 2
		g_two[04] 		:= thumb_3_max;
		g_two[05]		:= g_RestPos[05];	//	index 0
		g_two[06]		:= index_1_min;		//	index 1
		g_two[07]		:= index_2_min;		//	index 2
		g_two[08]		:= g_RestPos[08];	//	mid 0
		g_two[09]		:= mid_1_min;		//	mid 1
		g_two[10]		:= mid_2_min;		//	mid 2
		g_two[11]		:= g_RestPos[11];	//	ring 0
		g_two[12]		:= ring_1_max;		//	ring 1
		g_two[13]		:= ring_2_max;		//	ring 2
		g_two[14]		:= g_RestPos[14];	//	little 0
		g_two[15]		:= little_1_max;	//	little 1
		g_two[16]		:= little_2_max;	//	little 2
		g_two[17]		:= g_RestPos[17];	// wrist 0
		g_two[18]		:= g_RestPos[18];	// wrist 1
		
		//three
		g_three[01]		:= thumb_group_pos_2[0];	//thumb_0_max;	//	thumb 0
		g_three[02]		:= thumb_group_pos_2[1];	//thumb_1_max;	//	thumb 1
		g_three[03]		:= thumb_group_pos_2[2];	//thumb_2_max;	//	thumb 2
		g_three[04] 	:= thumb_3_max;
		g_three[05]		:= g_RestPos[05];	//	index 0
		g_three[06]		:= index_1_min;		//	index 1
		g_three[07]		:= index_2_min;		//	index 2
		g_three[08]		:= g_RestPos[08];	//	mid 0
		g_three[09]		:= mid_1_min;		//	mid 1
		g_three[10]		:= mid_2_min;		//	mid 2
		g_three[11]		:= g_RestPos[11];	//	ring 0
		g_three[12]		:= ring_1_min;		//	ring 1
		g_three[13]		:= ring_2_min;		//	ring 2
		g_three[14]		:= g_RestPos[14];	//	little 0
		g_three[15]		:= little_1_max;	//	little 1
		g_three[16]		:= little_2_max;	//	little 2
		g_three[17]		:= g_RestPos[17];	// wrist 0
		g_three[18]		:= g_RestPos[18];	// wrist 1
		
		
		//four
		g_four[01]		:= thumb_group_pos_2[0];	//thumb_0_max;	//	thumb 0
		g_four[02]		:= thumb_group_pos_2[1];	//thumb_1_max;	//	thumb 1
		g_four[03]		:= thumb_group_pos_2[2];	//thumb_2_max;	//	thumb 2
		g_four[04] 		:= thumb_3_max;
		g_four[05]		:= g_RestPos[05];	//	index 0
		g_four[06]		:= index_1_min;		//	index 1
		g_four[07]		:= index_2_min;		//	index 2
		g_four[08]		:= g_RestPos[08];	//	mid 0
		g_four[09]		:= mid_1_min;		//	mid 1
		g_four[10]		:= mid_2_min;		//	mid 2
		g_four[11]		:= g_RestPos[11];	//	ring 0
		g_four[12]		:= ring_1_min;		//	ring 1
		g_four[13]		:= ring_2_min;		//	ring 2
		g_four[14]		:= g_RestPos[14];	//	little 0
		g_four[15]		:= little_1_min;	//	little 1
		g_four[16]		:= little_2_min;	//	little 2
		g_four[17]		:= g_RestPos[17];	// wrist 0
		g_four[18]		:= g_RestPos[18];	// wrist 1
		
		
		//five
		g_five[01]		:= thumb_group_pos_0[0];	//thumb_0_min;	//	thumb 0
		g_five[02]		:= thumb_group_pos_0[1];	//thumb_1_min;	//	thumb 1
		g_five[03]		:= thumb_group_pos_0[2];	//thumb_2_min;	//	thumb 2
		g_five[04] 		:= thumb_3_min;
		g_five[05]		:= g_RestPos[05];	//	index 0
		g_five[06]		:= index_1_min;		//	index 1
		g_five[07]		:= index_2_min;		//	index 2
		g_five[08]		:= g_RestPos[08];	//	mid 0
		g_five[09]		:= mid_1_min;		//	mid 1
		g_five[10]		:= mid_2_min;		//	mid 2
		g_five[11]		:= g_RestPos[11];	//	ring 0
		g_five[12]		:= ring_1_min;		//	ring 1
		g_five[13]		:= ring_2_min;		//	ring 2
		g_five[14]		:= g_RestPos[14];	//	little 0
		g_five[15]		:= little_1_min;	//	little 1
		g_five[16]		:= little_2_min;	//	little 2
		g_five[17]		:= g_RestPos[17];	// wrist 0
		g_five[18]		:= g_RestPos[18];	// wrist 1
		
		
		//six
		g_six[01]		:= thumb_group_pos_0[0];	//thumb_0_min;	//	thumb 0
		g_six[02]		:= thumb_group_pos_0[1];	//thumb_1_min;	//	thumb 1
		g_six[03]		:= thumb_group_pos_0[2];	//thumb_2_min;	//	thumb 2
		g_six[04]		:= thumb_3_min;
		g_six[05]		:= g_RestPos[05];	//	index 0
		g_six[06]		:= index_1_max;		//	index 1
		g_six[07]		:= index_2_max;		//	index 2
		g_six[08]		:= g_RestPos[08];
		g_six[09]		:= mid_1_max;	//	mid 1
		g_six[10]		:= mid_2_max;	//	mid 2
		g_six[11]		:= g_RestPos[11];
		g_six[12]		:= ring_1_max;	//	ring 1
		g_six[13]		:= ring_2_max;	//	ring 2
		g_six[14]		:= g_RestPos[14];
		g_six[15]		:= little_1_min;	//	little 1
		g_six[16]		:= little_2_min;	//	little 2
		g_six[17]		:= g_RestPos[17];	// wrist 0
		g_six[18]		:= g_RestPos[18];	// wrist 1
		
		
		//plam
		g_plam[01]		:= thumb_group_pos_0[0];	//thumb_0_min;	//	thumb 0
		g_plam[02]		:= thumb_group_pos_0[1];	//thumb_1_min;	//	thumb 1
		g_plam[03]		:= thumb_group_pos_0[2];	//thumb_2_min;	//	thumb 2
		g_plam[04]		:= thumb_3_min;
		g_plam[05]		:= g_RestPos[05];
		g_plam[06]		:= index_1_min;	//	index 1
		g_plam[07]		:= index_2_min;	//	index 2
		g_plam[08]		:= g_RestPos[08];
		g_plam[09]		:= mid_1_min;	//	mid 1
		g_plam[10]		:= mid_2_min;	//	mid 2
		g_plam[11]		:= g_RestPos[11];
		g_plam[12]		:= ring_1_min;	//	ring 1
		g_plam[13]		:= ring_2_min;	//	ring 2
		g_plam[14]		:= g_RestPos[14];
		g_plam[15]		:= little_1_min;	//	little 1
		g_plam[16]		:= little_2_min;	//	little 2
		g_plam[17]		:= g_RestPos[17];	// wrist 0
		g_plam[18]		:= g_RestPos[18];	// wrist 1
		
		
		//fist
		g_fist[01]		:= thumb_group_pos_2[0];	//thumb_0_max;	//	thumb 0
		g_fist[02]		:= thumb_group_pos_2[1];	//thumb_1_max;	//	thumb 1
		g_fist[03]		:= thumb_group_pos_2[2];	//thumb_2_max;	//	thumb 2
		g_fist[04]		:= thumb_3_max;
		g_fist[05]		:= g_RestPos[05];
		g_fist[06]		:= index_1_max;	//	index 1
		g_fist[07]		:= index_2_max;	//	index 2
		g_fist[08]		:= g_RestPos[08];
		g_fist[09]		:= mid_1_max;	//	mid 1
		g_fist[10]		:= mid_2_max;	//	mid 2
		g_fist[11]		:= g_RestPos[11];
		g_fist[12]		:= ring_1_max;	//	ring 1
		g_fist[13]		:= ring_2_max;	//	ring 2
		g_fist[14]		:= g_RestPos[14];
		g_fist[15]		:= little_1_max;	//	little 1
		g_fist[16]		:= little_2_max;	//	little 2
		g_fist[17]		:= g_RestPos[17];	// wrist 0
		g_fist[18]		:= g_RestPos[18];	// wrist 1
		
		
		//thumb up
		g_thumbUp[01]		:= thumb_group_pos_0[0];	//thumb_0_min;	//	thumb 0
		g_thumbUp[02]		:= thumb_group_pos_0[1];	//thumb_1_min;	//	thumb 1
		g_thumbUp[03]		:= thumb_group_pos_0[2];	//thumb_2_min;	//	thumb 2
		g_thumbUp[04]		:= thumb_3_min;
		g_thumbUp[05]		:= g_RestPos[05];
		g_thumbUp[06]		:= index_1_max;	//	index 1
		g_thumbUp[07]		:= index_2_max;	//	index 2
		g_thumbUp[08]		:= g_RestPos[08];
		g_thumbUp[09]		:= mid_1_max;	//	mid 1
		g_thumbUp[10]		:= mid_2_max;	//	mid 2
		g_thumbUp[11]		:= g_RestPos[11];
		g_thumbUp[12]		:= ring_1_max;	//	ring 1
		g_thumbUp[13]		:= ring_2_max;	//	ring 2
		g_thumbUp[14]		:= g_RestPos[14];
		g_thumbUp[15]		:= little_1_max;	//	little 1
		g_thumbUp[16]		:= little_2_max;	//	little 2
		g_thumbUp[17]		:= g_RestPos[17];	// wrist 0
		g_thumbUp[18]		:= g_RestPos[18];	// wrist 1
		
		CycleMovTimes := 1;	// indecate the hand will move how many cycle.
		FOR i := 0 TO 10 DO
			DelayTime[i] := T#0S;
		END_FOR
		
		DelayTime[0]:= T#0S;
		CycleFingerMovPos[0] := g_RestPos;
		
		CASE Gesture OF
			Gesture_Type.Gesture_Type_none:
				state := -20;
				
			Gesture_Type.Gesture_Type_Num_1:
				SecFingerMovPos := FingerMovPos := g_one;
				
				FingerMovPos[01]	:= g_RestPos[01];	// thumb 0
				FingerMovPos[02]	:= g_RestPos[02];	// thumb 1
				FingerMovPos[03]	:= g_RestPos[03];	// thumb 2
				FingerMovPos[04]	:= g_RestPos[04];	// thumb 3
				
				CycleMovTimes := 2;
				CycleFingerMovPos[1] := FingerMovPos;
				CycleFingerMovPos[2] := SecFingerMovPos;

			Gesture_Type.Gesture_Type_Num_2:
				SecFingerMovPos := FingerMovPos := g_two;
				
				FingerMovPos[01]	:= g_RestPos[01];	// thumb 0
				FingerMovPos[02]	:= g_RestPos[02];	// thumb 1
				FingerMovPos[03]	:= g_RestPos[03];	// thumb 2
				FingerMovPos[04]	:= g_RestPos[04];	// thumb 3
				
				CycleMovTimes := 2;
				CycleFingerMovPos[1] := FingerMovPos;
				CycleFingerMovPos[2] := SecFingerMovPos;

			Gesture_Type.Gesture_Type_Num_3:
				SecFingerMovPos := FingerMovPos := g_three;
				
				FingerMovPos[01]	:= g_RestPos[01];	// thumb 0
				FingerMovPos[02]	:= g_RestPos[02];	// thumb 1
				FingerMovPos[03]	:= g_RestPos[03];	// thumb 2
				FingerMovPos[04]	:= g_RestPos[04];	// thumb 3
				
				CycleMovTimes := 2;
				CycleFingerMovPos[1] := FingerMovPos;
				CycleFingerMovPos[2] := SecFingerMovPos;

			Gesture_Type.Gesture_Type_Num_4:
				FingerMovPos := g_four;
				
				CycleFingerMovPos[1] := FingerMovPos;

			Gesture_Type.Gesture_Type_Num_5:
				FingerMovPos := g_five;
				
				CycleFingerMovPos[1] := FingerMovPos;

			Gesture_Type.Gesture_Type_Num_6:
				FingerMovPos := g_six;
				
				CycleFingerMovPos[1] := FingerMovPos;

			Gesture_Type.Gesture_Type_Fist:
				SecFingerMovPos := FingerMovPos := g_fist;
				
				FingerMovPos[01]	:= g_RestPos[01];	// thumb 0
				FingerMovPos[02]	:= g_RestPos[02];	// thumb 1
				FingerMovPos[03]	:= g_RestPos[03];	// thumb 2
				FingerMovPos[04]	:= g_RestPos[04];	// thumb 3
				
				CycleMovTimes := 2;
				CycleFingerMovPos[1] := FingerMovPos;
				CycleFingerMovPos[2] := SecFingerMovPos;
				
			Gesture_Type.Gesture_Type_Palm:
				FingerMovPos := g_plam;
				
				CycleFingerMovPos[1] := FingerMovPos;
				
			Gesture_Type.Gesture_Type_NoNoNo:
				ThdFingerMovPos := SecFingerMovPos := FingerMovPos := g_one;
				
				FingerMovPos[01]	:= g_RestPos[01];	// thumb 0
				FingerMovPos[02]	:= g_RestPos[02];	// thumb 1
				FingerMovPos[03]	:= g_RestPos[03];	// thumb 2
				FingerMovPos[04]	:= g_RestPos[04];	// thumb 3
				
				SecFingerMovPos[05] := index_0_max;
				SecFingerMovPos[17] := wrist_0_max;	// wrist 0
				
				ThdFingerMovPos[05] := -index_0_max;
				ThdFingerMovPos[17] := -wrist_0_max;	// wrist 0
				
				CycleMovTimes := 9;
				CycleFingerMovPos[1] := FingerMovPos;
				FOR i := 2 TO CycleMovTimes DO
					IF (i MOD 2) = 1 THEN
						CycleFingerMovPos[i] := SecFingerMovPos;
					ELSE
						CycleFingerMovPos[i] := ThdFingerMovPos;
					END_IF
				END_FOR
				
			Gesture_Type.Gesture_Type_ThumbUp:
				FingerMovPos := g_thumbup;
				
				CycleFingerMovPos[1] := FingerMovPos;
				
			Gesture_Type.Gesture_Type_ComeOnBaby:
			
				ThdFingerMovPos := SecFingerMovPos := FingerMovPos := g_one;
				
				FingerMovPos[01]	:= g_RestPos[01];	// thumb 0
				FingerMovPos[02]	:= g_RestPos[02];	// thumb 1
				FingerMovPos[03]	:= g_RestPos[03];	// thumb 2
				FingerMovPos[04]	:= g_RestPos[04];	// thumb 3
				
				SecFingerMovPos[06] := g_RestPos [06];
				SecFingerMovPos[07] := index_2_max;
				
				CycleMovTimes := 9;
				CycleFingerMovPos[1] := FingerMovPos;
				FOR i := 2 TO CycleMovTimes DO
					IF (i MOD 2) = 1 THEN
						CycleFingerMovPos[i] := SecFingerMovPos;
					ELSE
						CycleFingerMovPos[i] := ThdFingerMovPos;
					END_IF
				END_FOR
				
			Gesture_Type.Gesture_Type_FingerWave:
			
				ThdFingerMovPos := SecFingerMovPos := FingerMovPos := g_plam;
				
				SecFingerMovPos[01]	:= thumb_group_pos_1[00];	// thumb 0
				SecFingerMovPos[02]	:= thumb_group_pos_1[01];	// thumb 1
				SecFingerMovPos[03]	:= thumb_group_pos_1[02];	// thumb 2
				
				SecFingerMovPos[05]	:= index_0_max;	// thumb 2
				SecFingerMovPos[08]	:= mid_0_max;	// thumb 2
				SecFingerMovPos[11]	:= ring_0_max;	// thumb 2
				SecFingerMovPos[14]	:= little_0_max;	// thumb 2
				
				ThdFingerMovPos[01]	:= g_RestPos[01];	// thumb 0
				ThdFingerMovPos[02]	:= g_RestPos[02];	// thumb 1
				ThdFingerMovPos[03]	:= g_RestPos[03];	// thumb 2
				
				ThdFingerMovPos[05]	:= -index_0_max;	// thumb 2
				ThdFingerMovPos[08]	:= -mid_0_max;	// thumb 2
				ThdFingerMovPos[11]	:= -ring_0_max;	// thumb 2
				ThdFingerMovPos[14]	:= -little_0_max;	// thumb 2
				
				CycleMovTimes := 8;
				CycleFingerMovPos[1] := FingerMovPos;
				FOR i := 2 TO CycleMovTimes DO
					IF (i MOD 2) = 1 THEN
						CycleFingerMovPos[i] := SecFingerMovPos;
					ELSE
						CycleFingerMovPos[i] := ThdFingerMovPos;
					END_IF
				END_FOR
				
			Gesture_Type.Gesture_Type_Wave:
			
				SecFingerMovPos := FingerMovPos	:= g_two;
				
				FingerMovPos[17] := wrist_0_max;
				
				SecFingerMovPos[17] := -wrist_0_max;
				
				CycleMovTimes := 8;
				FOR i := 1 TO CycleMovTimes DO
					IF (i MOD 2) = 1 THEN
						CycleFingerMovPos[i] := FingerMovPos;
					ELSE
						CycleFingerMovPos[i] := SecFingerMovPos;
					END_IF
				END_FOR
					
			Gesture_Type.Gesture_Type_Nya:
			
				SecFingerMovPos := FingerMovPos	:= g_fist;
				
				FingerMovPos[18] := wrist_1_max;
				
				SecFingerMovPos[18] := - wrist_1_max;
				
				CycleMovTimes := 8;
				FOR i := 1 TO CycleMovTimes DO
					IF (i MOD 2) = 1 THEN
						CycleFingerMovPos[i] := FingerMovPos;
					ELSE
						CycleFingerMovPos[i] := SecFingerMovPos;
					END_IF
				END_FOR
				
			Gesture_Type.Gesture_Type_MovObj:
			(*
				G_MovObj_Muilt := 2;
				FingerMovPos	:= g_plam;
				SecFingerMovPos	:= g_fist;
				CycleMovTimes := 0;	// initialize
				
				CycleMovTimes := CycleMovTimes + 1;
				FingerMovPos[12] := -wrist_0_max;
				FingerMovPos[13] := wrist_1_max;
				// first mov, hand release go up left
				CycleFingerMovPos[CycleMovTimes] := FingerMovPos;
				//---
				
				CycleMovTimes := CycleMovTimes + 1;
				FingerMovPos[12] := wrist_0_max / G_MovObj_Muilt;
				FingerMovPos[13] := wrist_1_max;
				// sec mov, hand release go down left
				CycleFingerMovPos[CycleMovTimes] := FingerMovPos;
				//---
				
				CycleMovTimes := CycleMovTimes + 1;
				SecFingerMovPos[12] := wrist_0_max  / G_MovObj_Muilt;;
				SecFingerMovPos[13] := wrist_1_max;
				// third mov, hand grab at down left
				CycleFingerMovPos[CycleMovTimes] := SecFingerMovPos;
				//---
				
				CycleMovTimes := CycleMovTimes + 1;
				SecFingerMovPos[12] := -wrist_0_max;
				SecFingerMovPos[13] := wrist_1_max;
				// 4 mov, hand grab go up left
				CycleFingerMovPos[CycleMovTimes] := SecFingerMovPos;
				//---
				
				CycleMovTimes := CycleMovTimes + 1;
				SecFingerMovPos[12] := -wrist_0_max;
				SecFingerMovPos[13] := -wrist_1_max;
				// 5 mov, hand grab go up right
				CycleFingerMovPos[CycleMovTimes] := SecFingerMovPos;
				//---
				
				CycleMovTimes := CycleMovTimes + 1;
				SecFingerMovPos[12] := wrist_0_max / G_MovObj_Muilt;;
				SecFingerMovPos[13] := -wrist_1_max;
				// 6 mov, hand grab go down right
				CycleFingerMovPos[CycleMovTimes] := SecFingerMovPos;
				//---
				
				CycleMovTimes := CycleMovTimes + 1;
				FingerMovPos[12] := wrist_0_max / G_MovObj_Muilt;;
				FingerMovPos[13] := -wrist_1_max;
				// 7 mov, hand release at down right
				CycleFingerMovPos[CycleMovTimes] := FingerMovPos;
				//---
				
				CycleMovTimes := CycleMovTimes + 1;
				FingerMovPos[12] := -wrist_0_max;
				FingerMovPos[13] := -wrist_1_max;
				// 8 mov, hand release go up right
				DelayTime[CycleMovTimes] := T#3S;
				CycleFingerMovPos[CycleMovTimes] := FingerMovPos;
				//---
				
				CycleMovTimes := CycleMovTimes + 1;
				FingerMovPos[12] := wrist_0_max / G_MovObj_Muilt;;
				FingerMovPos[13] := -wrist_1_max;
				// 9 mov, hand release go down right
				CycleFingerMovPos[CycleMovTimes] := FingerMovPos;
				//---
				
				CycleMovTimes := CycleMovTimes + 1;
				SecFingerMovPos[12] := wrist_0_max / G_MovObj_Muilt;;
				SecFingerMovPos[13] := -wrist_1_max;
				// 10 mov, hand grab at down right
				CycleFingerMovPos[CycleMovTimes] := SecFingerMovPos;
				//---
				
				CycleMovTimes := CycleMovTimes + 1;
				SecFingerMovPos[12] := -wrist_0_max;
				SecFingerMovPos[13] := -wrist_1_max;
				// 11 mov, hand grab go up right
				CycleFingerMovPos[CycleMovTimes] := SecFingerMovPos;
				//---
				
				CycleMovTimes := CycleMovTimes + 1;
				SecFingerMovPos[12] := -wrist_0_max;
				SecFingerMovPos[13] := wrist_1_max;
				// 12 mov, hand grab go up left
				CycleFingerMovPos[CycleMovTimes] := SecFingerMovPos;
				//---
				
				CycleMovTimes := CycleMovTimes + 1;
				SecFingerMovPos[12] := wrist_0_max / G_MovObj_Muilt;;
				SecFingerMovPos[13] := wrist_1_max;
				// 13 mov, hand grab at down left
				CycleFingerMovPos[CycleMovTimes] := SecFingerMovPos;
				//---
				
				CycleMovTimes := CycleMovTimes + 1;
				FingerMovPos[12] := wrist_0_max / G_MovObj_Muilt;;
				FingerMovPos[13] := wrist_1_max;
				// 14 mov, hand release at down left
				CycleFingerMovPos[CycleMovTimes] := FingerMovPos;
				//---
				*)
		END_CASE
		
		
		i := 0;
		
		Give_Finger_Pos_Counter := 1;
		ArrayTotalNum := UINT_TO_INT(SIZEOF(CycleFingerMovPos)/SIZEOF(CycleFingerMovPos[1][1]));
		ArrayFirstRow := UINT_TO_INT((SIZEOF(CycleFingerMovPos)/SIZEOF(CycleFingerMovPos[1])));
		FOR MultiMov_for_counter := faxis TO laxis DO
			IF Give_Finger_Pos_Counter <= (ArrayTotalNum/ArrayFirstRow) THEN
				GivHandPos[MultiMov_for_counter] := CycleFingerMovPos[i][Give_Finger_Pos_Counter];
				Give_Finger_Pos_Counter := Give_Finger_Pos_Counter + 1;
			END_IF
		END_FOR
		MultiSingleMov(execute := FALSE);
		
		state := 40;
		
	40:
		IF (NOT enable) THEN
			State := 0;
		END_IF
		MultisingleMov(execute := TRUE, Axis_Mov_Indicator := AxisAllowToMov, axis_mov_pos := GivHandPos
			, vel := givenVel, acc :=givenAcc, dec := givenAcc, jerk := givenJerk, MoveMethod := 10);
		
		IF MultisingleMov.Done THEN
			IF DelayTime[i] > T#0S AND NOT DelayTimer.Q THEN
				DelayTimer(in := TRUE, pt := DelayTime[i]);
			ELSE
				DelayTimer(in := FALSE);
				i := i + 1;
				
				MultisingleMov(execute:= FALSE);
				Give_Finger_Pos_Counter := 1;
				FOR MultiMov_for_counter := faxis TO laxis DO
					IF Give_Finger_Pos_Counter <= (ArrayTotalNum/ArrayFirstRow) THEN
						GivHandPos[MultiMov_for_counter] := CycleFingerMovPos[i][Give_Finger_Pos_Counter];
						Give_Finger_Pos_Counter := Give_Finger_Pos_Counter + 1;
					END_IF
				END_FOR
			END_IF
		ELSIF MultisingleMov.error THEN
			state := -40;
		END_IF
		
		IF i > CycleMovTimes THEN
			state := 50;
		END_IF
	50:
		done := TRUE;
END_CASE

// end of the program

END_FUNCTION_BLOCK

// CODESYS_Control_x86_Arca_Control_SM/Application/Hand_Control_blocks/Hand_Gesture_Demo
FUNCTION_BLOCK Hand_Gesture_Demo
VAR_INPUT
	enable :BOOL;
	internal_hand_enable : BOOL;
	startMov :BOOL;
	ovr : INT;
	HandFirstAxis : BYTE;
	HandLastAxis : BYTE;
	HandAxisAllowToMov : ARRAY [0..17] OF BOOL;
END_VAR
VAR_OUTPUT
	IsEnabled : BOOL;
	IsMoving : BOOL;
	Current_Gesture : Gesture_type;
	err : BOOL;
	err_message : error_message;
END_VAR

VAR
	// state control
	cycleState : INT;	// state machine
	cycleCounter : INT;	// counte how many time already been done
	start_cycle : INT := 1;	// start cycle from a number
	total_cycle_time : INT := 14; //	max cycle time
	cycleTimer : ton;
	cycleDelayTime : TIME := T#2S;	// delay time between every gesture
	
	// hand powerOn
	powerHand : BOOL;
	powerOnHand : AuxAxis_PowerOn;
	_enabled : BOOL;
	
	// gestrure mov block
	GestureMov : Hand_Gesture;
	GestureType : ARRAY [1..16] OF Gesture_type;
END_VAR

// set gesture type
GestureType[1] := Gesture_type.Gesture_Type_Num_1;
GestureType[2] := Gesture_type.Gesture_Type_Num_2;
GestureType[3] := Gesture_type.Gesture_Type_Num_3;
GestureType[4] := Gesture_type.Gesture_Type_Num_4;
GestureType[5] := Gesture_type.Gesture_Type_Num_5;
GestureType[6] := Gesture_type.Gesture_Type_Num_6;
GestureType[7] := Gesture_type.Gesture_Type_Fist;
GestureType[8] := Gesture_type.Gesture_Type_Palm;
GestureType[9] := Gesture_type.Gesture_Type_ThumbUp;
GestureType[10] := Gesture_type.Gesture_Type_ComeOnBaby;
GestureType[11] := Gesture_type.Gesture_Type_wave;
GestureType[12] := Gesture_type.Gesture_Type_nya;
GestureType[13] := Gesture_type.Gesture_Type_NoNoNo;
GestureType[14] := Gesture_type.Gesture_Type_FingerWave;

//err
IF powerOnHand.Error OR GestureMov.Error THEN
	err := TRUE;
	IF powerOnHand.Error THEN
		err_message := powerOnHand.Err_Message;
	ELSIF GestureMov.Error THEN
		err_message := GestureMov.Err_Message;
	END_IF
ELSE
	err := FALSE;
	err_message := error_message.Err_None;
END_IF

// enable hand
IF internal_hand_enable THEN
	powerOnHand(enable := enable);
	_enabled := IsEnabled := powerOnHand.Done;
END_IF

IF NOT enable THEN
	cycleState := 0;
	isMoving := FALSE;
	cycleTimer(in := FALSE);	// reset timer
	GestureMov(Enable := FALSE);	// reset movement block
END_IF

CASE cycleState OF
	0: 
		// if block is enabled and order to move and (manager by internal power or by external power)
		IF enable AND startMov AND (NOT internal_hand_enable OR _enabled) THEN
			cycleCounter := start_cycle;	// set counter to start_cycle for gesture
			cycleState := 10;
		END_IF
	10:		GestureMov(Enable := TRUE, overfeed := ovr, Gesture := Current_Gesture := GestureType[cycleCounter], isMoving => isMoving
			, HandFirstAxis := HandFirstAxis, HandLastAxis:= HandLastAxis, HandAxisAllowToMov:= HandAxisAllowToMov);

		IF GestureMov.Done THEN
			cycleTimer(in := TRUE, pt:= cycleDelayTime);	// start timer for delay
			IF cycleTimer.Q THEN	// time reach
				cycleCounter := cycleCounter + 1;	// done and self add for next gesture
				cycleTimer(in := FALSE);	// reset timer
				GestureMov(Enable := FALSE);	// reset movement block
				IF cycleCounter <= total_cycle_time THEN
					cycleState := 10;	// if not reach total number then go back keep do next gesture
				ELSE
					cycleState := 0;	// if reach maximum then go back beginning
				END_IF
			END_IF
		END_IF
		
END_CASE

END_FUNCTION_BLOCK

// CODESYS_Control_x86_Arca_Control_SM/Application/TCPIP Control/TCPServerConnection
FUNCTION_BLOCK TCPServerConnection
VAR_INPUT
	Enable : BOOL;
	OutDataReady : BOOL;
	OutDataSize : CAA.SIZE;
	OutData :  ARRAY [0..255] OF BYTE;;
END_VAR
VAR_OUTPUT
	Err : BOOL;
	InDataReady : BOOL;
	InDataSize : CAA.SIZE;
	InData : STRING;
END_VAR
VAR
	TCPServer : NBS.TCP_Server;
	IP_Addr : NBS.IP_ADDR := (sAddr :='192.168.80.240');
	Port: UINT := 23; // TCP/IP port
	TCPS_Err : BOOL := FALSE;
	TCPS_Err_Mssage : NBS.ERROR;
	
	TCPS_Connection : NBS.TCP_Connection;
	
	ServerRead : NBS.TCP_Read;
	ServerSend : NBS.TCP_Write;
	
	Hendle_enable :BOOL;
	Some_Connect_In : BOOL;
	
	// message out
	_OutDataSize : CAA.SIZE;
	debug : BOOL;
	testTXT :STRING := '0123456';
	testByte : ARRAY [0..5] OF BYTE := [40,12,41,40,10,41];
	ddone, deErr, dxErr : BOOL;
END_VAR

// initialize TCP server
TCPServer(xEnable := Enable, ipAddr := IP_Addr, uiPort := Port, xError => TCPS_Err, eError => TCPS_Err_Mssage);

// send handle after there are some client connect 
TCPS_Connection(xEnable := Hendle_enable, hServer := TCPServer.hServer);

// enable handle after tcp server is online, up below command is insure if there is a client disconnect, the command will be turn off one cycle
IF TCPServer.xBusy AND NOT Hendle_enable THEN
	Hendle_enable := TRUE;
ELSIF NOT TCPServer.xBusy AND Hendle_enable THEN
	Hendle_enable := FALSE;
END_IF

// some one connect in
IF TCPS_Connection.xActive THEN
	Some_Connect_In := TRUE;
END_IF

// health check, if connection broken then turn off handle to wait next connection
IF Some_Connect_In AND NOT TCPS_Connection.xActive THEN
	Some_Connect_In := Hendle_enable := FALSE;
END_IF

// receive data from client
ServerRead(xEnable := TCPS_Connection.xActive, hConnection := TCPS_Connection.hConnection
	, szSize := SIZEOF(InData)
	, pData := ADR(InData)
	, szCount => InDataSize
	, xReady => InDataReady	// when new data comes this flag will be true in one cycle
	);

	
// send data to client
IF OutDataSize > 0 THEN
	_OutDataSize := OutDataSize;
ELSE
	_OutDataSize := SIZEOF(OutData);
END_IF

IF outdataReady THEN
	debug := TRUE;
END_IF

ServerSend(xExecute := OutDataReady, hConnection := TCPS_Connection.hConnection, szSize := _OutDataSize, pData := ADR(OutData), udiTimeOut := 1000
	, xError => dxErr, xDone => ddone);

END_FUNCTION_BLOCK

